C05477=1176.105,271.034,-67.370,-177.096,7.526,148.586
C05478=1176.109,270.786,-67.343,-177.099,7.524,148.586
C05479=1176.114,270.537,-67.314,-177.101,7.521,148.586
C05480=1176.118,270.290,-67.286,-177.104,7.518,148.586
C05481=1176.123,270.041,-67.257,-177.107,7.515,148.586
C05482=1176.127,269.793,-67.230,-177.109,7.513,148.586
C05483=1176.131,269.544,-67.202,-177.112,7.510,148.586
C05484=1176.135,269.295,-67.173,-177.114,7.507,148.586
C05485=1176.140,269.047,-67.145,-177.117,7.504,148.586
C05486=1176.144,268.799,-67.116,-177.119,7.502,148.586
C05487=1176.149,268.551,-67.088,-177.122,7.499,148.586
C05488=1176.153,268.302,-67.060,-177.125,7.496,148.586
C05489=1176.157,268.054,-67.032,-177.128,7.493,148.586
C05490=1176.162,267.806,-67.004,-177.130,7.491,148.586
C05491=1176.166,267.557,-66.975,-177.132,7.488,148.586
C05492=1176.171,267.309,-66.948,-177.136,7.485,148.587
C05493=1176.174,267.061,-66.920,-177.138,7.483,148.587
C05494=1176.180,266.812,-66.892,-177.141,7.480,148.587
C05495=1176.183,266.563,-66.864,-177.143,7.477,148.587
C05496=1176.188,266.315,-66.836,-177.146,7.474,148.587
C05497=1176.192,266.067,-66.807,-177.148,7.472,148.587
C05498=1176.197,265.819,-66.779,-177.151,7.469,148.587
C05499=1176.200,265.570,-66.751,-177.154,7.466,148.587
C05500=1176.206,265.321,-66.724,-177.156,7.463,148.587
C05501=1176.210,265.073,-66.696,-177.159,7.461,148.587
C05502=1176.214,264.825,-66.668,-177.161,7.458,148.587
C05503=1176.218,264.577,-66.640,-177.164,7.455,148.587
C05504=1176.223,264.327,-66.612,-177.167,7.453,148.588
C05505=1176.227,264.080,-66.584,-177.169,7.450,148.588
C05506=1176.232,263.832,-66.556,-177.172,7.447,148.588
C05507=1176.235,263.583,-66.528,-177.174,7.445,148.588
C05508=1176.241,263.334,-66.501,-177.177,7.442,148.588
C05509=1176.245,263.086,-66.472,-177.180,7.439,148.588
C05510=1176.249,262.838,-66.445,-177.183,7.436,148.588
C05511=1176.254,262.565,-66.414,-177.185,7.433,148.588
C05512=1176.259,262.292,-66.384,-177.189,7.430,148.588
C05513=1176.264,262.019,-66.353,-177.191,7.427,148.588
C05514=1176.268,261.745,-66.322,-177.194,7.424,148.588
C05515=1176.273,261.497,-66.295,-177.197,7.421,148.589
C05516=1176.277,261.249,-66.267,-177.199,7.419,148.589
C05517=1176.281,261.000,-66.239,-177.202,7.417,148.589
C05518=1176.286,260.752,-66.212,-177.205,7.414,148.589
C05519=1176.290,260.504,-66.184,-177.207,7.412,148.589
C05520=1176.295,260.254,-66.156,-177.210,7.409,148.589
C05521=1176.299,260.007,-66.129,-177.213,7.406,148.589
C05522=1176.304,259.758,-66.102,-177.215,7.403,148.589
C05523=1176.308,259.509,-66.073,-177.217,7.400,148.589
C05524=1176.312,259.261,-66.046,-177.221,7.398,148.590
C05525=1176.317,259.013,-66.019,-177.223,7.396,148.590
C05526=1176.321,258.765,-65.992,-177.226,7.393,148.590
C05527=1176.325,258.516,-65.963,-177.228,7.390,148.590
C05528=1176.330,258.268,-65.936,-177.231,7.388,148.590
C05529=1176.334,258.019,-65.909,-177.233,7.385,148.590
C05530=1176.338,257.770,-65.881,-177.236,7.382,148.590
C05531=1176.343,257.522,-65.854,-177.239,7.380,148.590
C05532=1176.347,257.274,-65.826,-177.241,7.377,148.590
C05533=1176.352,257.026,-65.799,-177.244,7.374,148.590
C05534=1176.356,256.776,-65.772,-177.246,7.372,148.590
C05535=1176.360,256.529,-65.744,-177.249,7.369,148.591
C05536=1176.365,256.280,-65.717,-177.252,7.366,148.591
C05537=1176.369,256.032,-65.690,-177.254,7.364,148.591
C05538=1176.373,255.783,-65.662,-177.257,7.361,148.591
C05539=1176.378,255.534,-65.635,-177.260,7.358,148.591
C05540=1176.382,255.286,-65.608,-177.262,7.356,148.591
C05541=1176.387,255.038,-65.580,-177.265,7.353,148.591
C05542=1176.391,254.789,-65.552,-177.268,7.350,148.591
C05543=1176.396,254.540,-65.525,-177.270,7.348,148.592
C05544=1176.400,254.292,-65.498,-177.273,7.345,148.592
C05545=1176.405,254.044,-65.471,-177.276,7.342,148.592
C05546=1176.409,253.796,-65.444,-177.278,7.340,148.592
C05547=1176.413,253.546,-65.416,-177.281,7.337,148.592
C05548=1176.418,253.298,-65.389,-177.283,7.335,148.592
C05549=1176.422,253.050,-65.363,-177.286,7.332,148.592
C05550=1176.426,252.801,-65.336,-177.289,7.330,148.592
C05551=1176.431,252.553,-65.308,-177.291,7.327,148.593
C05552=1176.436,252.305,-65.281,-177.294,7.325,148.593
C05553=1176.440,252.056,-65.253,-177.297,7.322,148.593
C05554=1176.444,251.807,-65.226,-177.299,7.319,148.593
C05555=1176.449,251.559,-65.199,-177.302,7.317,148.593
C05556=1176.453,251.310,-65.173,-177.304,7.315,148.593
C05557=1176.457,251.062,-65.146,-177.307,7.312,148.593
C05558=1176.462,250.813,-65.119,-177.310,7.309,148.593
C05559=1176.467,250.565,-65.091,-177.313,7.307,148.594
C05560=1176.471,250.316,-65.064,-177.315,7.304,148.594
C05561=1176.475,250.068,-65.038,-177.318,7.301,148.594
C05562=1176.479,249.819,-65.011,-177.320,7.299,148.594
C05563=1176.484,249.571,-64.983,-177.323,7.296,148.594
C05564=1176.489,249.322,-64.956,-177.326,7.294,148.594
C05565=1176.493,249.074,-64.930,-177.328,7.291,148.594
C05566=1176.497,248.825,-64.903,-177.331,7.288,148.594
C05567=1176.502,248.577,-64.876,-177.334,7.286,148.595
C05568=1176.507,248.328,-64.849,-177.337,7.283,148.595
C05569=1176.510,248.080,-64.822,-177.339,7.281,148.595
C05570=1176.515,247.831,-64.795,-177.342,7.278,148.595
C05571=1176.519,247.583,-64.768,-177.345,7.276,148.595
C05572=1176.523,247.334,-64.741,-177.347,7.273,148.595
C05573=1176.528,247.086,-64.714,-177.350,7.270,148.595
C05574=1176.533,246.837,-64.688,-177.352,7.269,148.596
C05575=1176.537,246.589,-64.661,-177.355,7.266,148.596
C05576=1176.541,246.340,-64.634,-177.358,7.263,148.596
C05577=1176.546,246.092,-64.607,-177.360,7.261,148.596
C05578=1176.550,245.843,-64.581,-177.363,7.258,148.596
C05579=1176.555,245.595,-64.554,-177.365,7.256,148.596
C05580=1176.560,245.346,-64.527,-177.368,7.253,148.596
C05581=1176.563,245.098,-64.501,-177.371,7.251,148.597
C05582=1176.568,244.849,-64.474,-177.373,7.248,148.597
C05583=1176.572,244.601,-64.447,-177.376,7.245,148.597
C05584=1176.577,244.352,-64.421,-177.379,7.243,148.597
C05585=1176.582,244.103,-64.394,-177.382,7.240,148.597
C05586=1176.586,243.855,-64.368,-177.384,7.238,148.597
C05587=1176.590,243.607,-64.341,-177.387,7.235,148.597
C05588=1176.594,243.358,-64.315,-177.389,7.233,148.598
C05589=1176.599,243.109,-64.288,-177.392,7.230,148.598
C05590=1176.603,242.861,-64.261,-177.395,7.228,148.598
C05591=1176.608,242.612,-64.235,-177.397,7.226,148.598
C05592=1176.612,242.364,-64.208,-177.400,7.223,148.598
C05593=1176.617,242.115,-64.182,-177.403,7.221,148.598
C05594=1176.622,241.866,-64.155,-177.405,7.218,148.598
C05595=1176.625,241.618,-64.129,-177.408,7.216,148.599
C05596=1176.630,241.369,-64.102,-177.411,7.213,148.599
C05597=1176.634,241.121,-64.076,-177.413,7.211,148.599
C05598=1176.639,240.872,-64.050,-177.416,7.208,148.599
C05599=1176.643,240.623,-64.023,-177.419,7.205,148.599
C05600=1176.647,240.375,-63.997,-177.421,7.203,148.599
C05601=1176.653,240.127,-63.970,-177.424,7.200,148.600
C05602=1176.657,239.878,-63.945,-177.427,7.198,148.600
C05603=1176.662,239.630,-63.918,-177.429,7.195,148.600
C05604=1176.666,239.381,-63.892,-177.432,7.194,148.600
C05605=1176.670,239.132,-63.865,-177.435,7.191,148.600
C05606=1176.675,238.883,-63.839,-177.437,7.189,148.600
C05607=1176.679,238.635,-63.813,-177.440,7.186,148.601
C05608=1176.684,238.386,-63.786,-177.442,7.184,148.601
C05609=1176.687,238.138,-63.760,-177.445,7.181,148.601
C05610=1176.692,237.889,-63.733,-177.448,7.179,148.601
C05611=1176.697,237.641,-63.708,-177.450,7.176,148.601
C05612=1176.701,237.393,-63.682,-177.453,7.174,148.602
C05613=1176.706,237.143,-63.655,-177.456,7.171,148.602
C05614=1176.710,236.895,-63.629,-177.459,7.168,148.602
C05615=1176.715,236.623,-63.601,-177.461,7.166,148.602
C05616=1176.720,236.352,-63.571,-177.464,7.164,148.602
C05617=1176.725,236.080,-63.543,-177.467,7.161,148.602
C05618=1176.730,235.809,-63.515,-177.470,7.158,148.603
C05619=1176.735,235.560,-63.489,-177.473,7.156,148.603
C05620=1176.739,235.311,-63.463,-177.475,7.153,148.603
C05621=1176.743,235.063,-63.437,-177.478,7.151,148.603
C05622=1176.748,234.814,-63.410,-177.481,7.148,148.603
C05623=1176.752,234.565,-63.384,-177.483,7.147,148.604
C05624=1176.757,234.317,-63.359,-177.486,7.144,148.604
C05625=1176.761,234.068,-63.333,-177.488,7.141,148.604
C05626=1176.766,233.820,-63.306,-177.492,7.139,148.604
C05627=1176.770,233.571,-63.280,-177.494,7.137,148.604
C05628=1176.775,233.323,-63.255,-177.497,7.134,148.604
C05629=1176.779,233.074,-63.229,-177.499,7.132,148.605
C05630=1176.784,232.825,-63.203,-177.502,7.129,148.605
C05631=1176.788,232.576,-63.177,-177.505,7.127,148.605
C05632=1176.792,232.328,-63.151,-177.508,7.125,148.605
C05633=1176.797,232.080,-63.125,-177.510,7.122,148.605
C05634=1176.801,231.831,-63.100,-177.513,7.119,148.605
C05635=1176.805,231.582,-63.074,-177.515,7.118,148.606
C05636=1176.810,231.333,-63.047,-177.518,7.115,148.606
C05637=1176.815,231.085,-63.022,-177.521,7.113,148.606
C05638=1176.819,230.836,-62.996,-177.523,7.110,148.606
C05639=1176.823,230.587,-62.971,-177.526,7.108,148.607
C05640=1176.828,230.339,-62.945,-177.529,7.105,148.607
C05641=1176.833,230.091,-62.919,-177.532,7.103,148.607
C05642=1176.837,229.841,-62.893,-177.534,7.100,148.607
C05643=1176.842,229.593,-62.867,-177.537,7.099,148.607
C05644=1176.847,229.345,-62.842,-177.540,7.096,148.607
C05645=1176.851,229.096,-62.816,-177.542,7.094,148.608
C05646=1176.855,228.847,-62.790,-177.545,7.092,148.608
C05647=1176.860,228.599,-62.765,-177.548,7.089,148.608
C05648=1176.864,228.350,-62.739,-177.550,7.087,148.608
C05649=1176.868,228.101,-62.714,-177.553,7.084,148.608
C05650=1176.873,227.853,-62.688,-177.555,7.082,148.609
C05651=1176.877,227.604,-62.662,-177.558,7.079,148.609
C05652=1176.882,227.355,-62.637,-177.561,7.077,148.609
C05653=1176.886,227.107,-62.611,-177.564,7.074,148.609
C05654=1176.891,226.858,-62.586,-177.566,7.073,148.610
C05655=1176.895,226.609,-62.561,-177.569,7.070,148.610
C05656=1176.900,226.361,-62.535,-177.572,7.068,148.610
C05657=1176.904,226.112,-62.509,-177.574,7.066,148.610
C05658=1176.908,225.863,-62.484,-177.577,7.063,148.610
C05659=1176.913,225.615,-62.458,-177.579,7.061,148.610
C05660=1176.918,225.366,-62.433,-177.582,7.058,148.611
C05661=1176.922,225.117,-62.407,-177.585,7.056,148.611
C05662=1176.927,224.869,-62.382,-177.588,7.054,148.611
C05663=1176.931,224.620,-62.356,-177.590,7.052,148.611
C05664=1176.936,224.371,-62.332,-177.593,7.050,148.612
C05665=1176.940,224.123,-62.306,-177.596,7.047,148.612
C05666=1176.945,223.874,-62.280,-177.598,7.045,148.612
C05667=1176.949,223.626,-62.255,-177.601,7.042,148.612
C05668=1176.954,223.376,-62.230,-177.603,7.040,148.612
C05669=1176.959,223.128,-62.204,-177.607,7.037,148.613
C05670=1176.963,222.879,-62.179,-177.609,7.035,148.613
C05671=1176.967,222.631,-62.155,-177.612,7.034,148.613
C05672=1176.972,222.382,-62.129,-177.614,7.031,148.613
C05673=1176.976,222.133,-62.103,-177.617,7.029,148.614
C05674=1176.981,221.885,-62.078,-177.620,7.026,148.614
C05675=1176.985,221.636,-62.053,-177.622,7.024,148.614
C05676=1176.990,221.387,-62.028,-177.625,7.022,148.614
C05677=1176.995,221.138,-62.002,-177.628,7.019,148.614
C05678=1176.999,220.891,-61.977,-177.630,7.017,148.615
C05679=1177.003,220.641,-61.952,-177.633,7.014,148.615
C05680=1177.008,220.393,-61.927,-177.636,7.013,148.615
C05681=1177.013,220.144,-61.902,-177.638,7.011,148.615
C05682=1177.017,219.896,-61.877,-177.641,7.008,148.616
C05683=1177.021,219.646,-61.852,-177.644,7.006,148.616
C05684=1177.026,219.398,-61.827,-177.647,7.003,148.616
C05685=1177.031,219.149,-61.802,-177.649,7.001,148.616
C05686=1177.035,218.901,-61.776,-177.652,6.999,148.616
C05687=1177.040,218.651,-61.751,-177.655,6.997,148.617
C05688=1177.044,218.404,-61.726,-177.657,6.994,148.617
C05689=1177.048,218.154,-61.701,-177.660,6.992,148.617
C05690=1177.053,217.906,-61.676,-177.663,6.990,148.618
C05691=1177.057,217.657,-61.652,-177.665,6.988,148.618
C05692=1177.062,217.408,-61.627,-177.668,6.985,148.618
C05693=1177.066,217.159,-61.601,-177.670,6.983,148.618
C05694=1177.072,216.911,-61.577,-177.674,6.981,148.618
C05695=1177.075,216.662,-61.551,-177.676,6.979,148.619
C05696=1177.080,216.413,-61.527,-177.678,6.977,148.619
C05697=1177.085,216.164,-61.502,-177.682,6.974,148.619
C05698=1177.089,215.916,-61.477,-177.684,6.972,148.619
C05699=1177.093,215.667,-61.452,-177.687,6.970,148.620
C05700=1177.098,215.418,-61.427,-177.690,6.967,148.620
C05701=1177.103,215.170,-61.402,-177.692,6.965,148.620
C05702=1177.107,214.921,-61.377,-177.695,6.964,148.620
C05703=1177.112,214.672,-61.353,-177.697,6.961,148.620
C05704=1177.116,214.423,-61.328,-177.700,6.959,148.621
C05705=1177.121,214.175,-61.303,-177.703,6.956,148.621
C05706=1177.125,213.927,-61.279,-177.705,6.954,148.621
C05707=1177.130,213.677,-61.254,-177.708,6.952,148.622
C05708=1177.135,213.428,-61.229,-177.711,6.949,148.622
C05709=1177.138,213.180,-61.204,-177.714,6.947,148.622
C05710=1177.144,212.931,-61.179,-177.716,6.946,148.622
C05711=1177.148,212.683,-61.155,-177.719,6.943,148.622
C05712=1177.152,212.433,-61.130,-177.722,6.941,148.623
C05713=1177.157,212.185,-61.106,-177.724,6.939,148.623
C05714=1177.162,211.936,-61.081,-177.727,6.936,148.623
C05715=1177.165,211.688,-61.056,-177.730,6.934,148.623
C05716=1177.171,211.439,-61.032,-177.732,6.932,148.624
C05717=1177.176,211.190,-61.007,-177.735,6.930,148.624
C05718=1177.180,210.941,-60.982,-177.738,6.928,148.624
C05719=1177.185,210.671,-60.956,-177.741,6.925,148.625
C05720=1177.190,210.401,-60.929,-177.743,6.923,148.625
C05721=1177.195,210.129,-60.903,-177.746,6.920,148.625
C05722=1177.200,209.859,-60.876,-177.750,6.918,148.625
C05723=1177.204,209.611,-60.852,-177.752,6.916,148.626
C05724=1177.209,209.361,-60.827,-177.755,6.914,148.626
C05725=1177.213,209.113,-60.803,-177.758,6.911,148.626
C05726=1177.218,208.864,-60.778,-177.760,6.910,148.626
C05727=1177.222,208.615,-60.754,-177.763,6.907,148.627
C05728=1177.226,208.367,-60.730,-177.765,6.906,148.627
C05729=1177.232,208.118,-60.705,-177.768,6.903,148.627
C05730=1177.236,207.869,-60.681,-177.771,6.901,148.627
C05731=1177.241,207.620,-60.656,-177.773,6.899,148.628
C05732=1177.245,207.372,-60.632,-177.776,6.896,148.628
C05733=1177.250,207.123,-60.607,-177.779,6.894,148.628
C05734=1177.254,206.874,-60.583,-177.781,6.893,148.628
C05735=1177.258,206.625,-60.559,-177.785,6.890,148.629
C05736=1177.263,206.377,-60.534,-177.787,6.888,148.629
C05737=1177.268,206.128,-60.510,-177.790,6.886,148.629
C05738=1177.272,205.879,-60.486,-177.793,6.883,148.630
C05739=1177.277,205.630,-60.461,-177.795,6.881,148.630
C05740=1177.281,205.381,-60.437,-177.798,6.879,148.630
C05741=1177.286,205.133,-60.413,-177.800,6.878,148.630
C05742=1177.291,204.884,-60.389,-177.803,6.875,148.630
C05743=1177.296,204.635,-60.365,-177.806,6.873,148.631
C05744=1177.299,204.386,-60.341,-177.808,6.871,148.631
C05745=1177.305,204.137,-60.316,-177.811,6.868,148.631
C05746=1177.309,203.889,-60.292,-177.814,6.866,148.632
C05747=1177.313,203.641,-60.268,-177.816,6.865,148.632
C05748=1177.318,203.392,-60.245,-177.819,6.862,148.632
C05749=1177.323,203.142,-60.220,-177.822,6.860,148.632
C05750=1177.327,202.894,-60.196,-177.825,6.858,148.633
C05751=1177.332,202.645,-60.172,-177.827,6.856,148.633
C05752=1177.336,202.396,-60.148,-177.830,6.853,148.633
C05753=1177.341,202.148,-60.123,-177.833,6.852,148.633
C05754=1177.345,201.898,-60.100,-177.835,6.850,148.634
C05755=1177.350,201.649,-60.076,-177.838,6.848,148.634
C05756=1177.354,201.401,-60.052,-177.841,6.845,148.634
C05757=1177.360,201.152,-60.028,-177.843,6.843,148.635
C05758=1177.364,200.903,-60.004,-177.846,6.841,148.635
C05759=1177.368,200.655,-59.979,-177.848,6.839,148.635
C05760=1177.373,200.406,-59.956,-177.852,6.837,148.635
C05761=1177.377,200.157,-59.932,-177.854,6.835,148.636
C05762=1177.381,199.908,-59.908,-177.856,6.833,148.636
C05763=1177.387,199.659,-59.884,-177.859,6.831,148.636
C05764=1177.391,199.410,-59.860,-177.862,6.828,148.637
C05765=1177.396,199.161,-59.836,-177.865,6.827,148.637
C05766=1177.400,198.913,-59.812,-177.867,6.824,148.637
C05767=1177.405,198.664,-59.789,-177.870,6.823,148.637
C05768=1177.409,198.416,-59.765,-177.873,6.820,148.638
C05769=1177.414,198.167,-59.741,-177.876,6.818,148.638
C05770=1177.418,197.918,-59.717,-177.878,6.816,148.638
C05771=1177.423,197.668,-59.693,-177.881,6.814,148.639
C05772=1177.428,197.419,-59.670,-177.884,6.812,148.639
C05773=1177.432,197.171,-59.645,-177.887,6.810,148.639
C05774=1177.437,196.922,-59.622,-177.889,6.808,148.639
C05775=1177.441,196.673,-59.598,-177.891,6.806,148.640
C05776=1177.446,196.424,-59.575,-177.895,6.803,148.640
C05777=1177.450,196.176,-59.551,-177.897,6.802,148.640
C05778=1177.455,195.927,-59.527,-177.899,6.800,148.640
C05779=1177.460,195.678,-59.504,-177.902,6.798,148.641
C05780=1177.464,195.429,-59.480,-177.905,6.795,148.641
C05781=1177.469,195.180,-59.456,-177.908,6.793,148.642
C05782=1177.474,194.931,-59.433,-177.910,6.791,148.642
C05783=1177.478,194.683,-59.409,-177.913,6.789,148.642
C05784=1177.483,194.434,-59.386,-177.916,6.788,148.642
C05785=1177.487,194.185,-59.362,-177.919,6.785,148.643
C05786=1177.492,193.936,-59.338,-177.921,6.783,148.643
C05787=1177.497,193.687,-59.315,-177.924,6.781,148.643
C05788=1177.501,193.438,-59.292,-177.926,6.779,148.643
C05789=1177.506,193.189,-59.268,-177.929,6.778,148.644
C05790=1177.510,192.941,-59.244,-177.932,6.775,148.644
C05791=1177.515,192.692,-59.221,-177.934,6.773,148.644
C05792=1177.520,192.443,-59.197,-177.937,6.771,148.645
C05793=1177.524,192.194,-59.174,-177.940,6.769,148.645
C05794=1177.529,191.945,-59.150,-177.943,6.767,148.645
C05795=1177.533,191.697,-59.127,-177.946,6.765,148.646
C05796=1177.537,191.448,-59.104,-177.948,6.763,148.646
C05797=1177.542,191.199,-59.080,-177.951,6.761,148.646
C05798=1177.547,190.949,-59.057,-177.953,6.759,148.647
C05799=1177.552,190.700,-59.034,-177.957,6.757,148.647
C05800=1177.556,190.452,-59.010,-177.959,6.755,148.647
C05801=1177.561,190.203,-58.986,-177.961,6.753,148.647
C05802=1177.566,189.955,-58.963,-177.964,6.751,148.648
C05803=1177.571,189.706,-58.940,-177.967,6.749,148.648
C05804=1177.575,189.457,-58.917,-177.969,6.747,148.648
C05805=1177.579,189.208,-58.894,-177.973,6.745,148.649
C05806=1177.584,188.959,-58.870,-177.975,6.743,148.649
C05807=1177.589,188.710,-58.847,-177.978,6.741,148.649
C05808=1177.593,188.461,-58.824,-177.980,6.739,148.650
C05809=1177.597,188.212,-58.801,-177.983,6.737,148.650
C05810=1177.602,187.963,-58.778,-177.986,6.735,148.650
C05811=1177.607,187.714,-58.754,-177.988,6.733,148.650
C05812=1177.612,187.466,-58.731,-177.991,6.731,148.651
C05813=1177.617,187.217,-58.708,-177.994,6.729,148.651
C05814=1177.621,186.968,-58.685,-177.996,6.727,148.651
C05815=1177.625,186.719,-58.662,-177.999,6.725,148.652
C05816=1177.630,186.470,-58.638,-178.002,6.723,148.652
C05817=1177.635,186.221,-58.615,-178.004,6.721,148.652
C05818=1177.639,185.972,-58.592,-178.007,6.719,148.653
C05819=1177.644,185.724,-58.569,-178.010,6.717,148.653
C05820=1177.649,185.475,-58.546,-178.012,6.715,148.653
C05821=1177.653,185.226,-58.523,-178.015,6.714,148.654
C05822=1177.658,184.976,-58.501,-178.018,6.712,148.654
C05823=1177.663,184.707,-58.475,-178.021,6.709,148.654
C05824=1177.667,184.438,-58.450,-178.024,6.707,148.655
C05825=1177.673,184.168,-58.425,-178.027,6.705,148.655
C05826=1177.678,183.898,-58.400,-178.030,6.703,148.655
C05827=1177.682,183.650,-58.378,-178.032,6.701,148.656
C05828=1177.687,183.400,-58.354,-178.035,6.699,148.656
C05829=1177.692,183.152,-58.332,-178.038,6.697,148.656
C05830=1177.696,182.903,-58.309,-178.040,6.695,148.657
C05831=1177.701,182.654,-58.286,-178.043,6.693,148.657
C05832=1177.706,182.405,-58.262,-178.046,6.691,148.657
C05833=1177.710,182.155,-58.240,-178.048,6.689,148.658
C05834=1177.715,181.907,-58.217,-178.051,6.687,148.658
C05835=1177.719,181.658,-58.195,-178.053,6.686,148.658
C05836=1177.724,181.409,-58.171,-178.056,6.684,148.659
C05837=1177.728,181.160,-58.149,-178.059,6.681,148.659
C05838=1177.733,180.912,-58.126,-178.062,6.679,148.659
C05839=1177.738,180.663,-58.103,-178.065,6.678,148.660
C05840=1177.742,180.413,-58.081,-178.067,6.676,148.660
C05841=1177.747,180.164,-58.057,-178.070,6.674,148.660
C05842=1177.752,179.916,-58.035,-178.072,6.672,148.660
C05843=1177.757,179.667,-58.012,-178.075,6.670,148.661
C05844=1177.761,179.418,-57.990,-178.078,6.668,148.661
C05845=1177.765,179.169,-57.966,-178.081,6.666,148.662
C05846=1177.770,178.920,-57.945,-178.083,6.664,148.662
C05847=1177.775,178.671,-57.921,-178.086,6.662,148.662
C05848=1177.779,178.422,-57.899,-178.089,6.661,148.663
C05849=1177.784,178.173,-57.876,-178.091,6.659,148.663
C05850=1177.789,177.924,-57.854,-178.094,6.657,148.663
C05851=1177.793,177.675,-57.831,-178.096,6.655,148.663
C05852=1177.798,177.427,-57.808,-178.099,6.653,148.664
C05853=1177.803,177.177,-57.786,-178.102,6.651,148.664
C05854=1177.807,176.929,-57.763,-178.104,6.650,148.665
C05855=1177.813,176.680,-57.741,-178.108,6.647,148.665
C05856=1177.817,176.431,-57.718,-178.110,6.645,148.665
C05857=1177.821,176.182,-57.696,-178.113,6.643,148.666
C05858=1177.826,175.933,-57.674,-178.116,6.642,148.666
C05859=1177.830,175.684,-57.651,-178.118,6.640,148.666
C05860=1177.835,175.434,-57.628,-178.121,6.638,148.666
C05861=1177.840,175.186,-57.606,-178.123,6.636,148.667
C05862=1177.845,174.937,-57.583,-178.126,6.634,148.667
C05863=1177.849,174.688,-57.560,-178.129,6.632,148.668
C05864=1177.854,174.439,-57.539,-178.131,6.631,148.668
C05865=1177.859,174.190,-57.516,-178.134,6.629,148.668
C05866=1177.863,173.941,-57.493,-178.137,6.627,148.669
C05867=1177.868,173.692,-57.472,-178.140,6.624,148.669
C05868=1177.872,173.443,-57.448,-178.143,6.623,148.669
C05869=1177.877,173.195,-57.427,-178.145,6.621,148.670
C05870=1177.881,172.945,-57.405,-178.148,6.619,148.670
C05871=1177.886,172.696,-57.381,-178.151,6.617,148.670
C05872=1177.891,172.448,-57.359,-178.153,6.616,148.671
C05873=1177.895,172.198,-57.337,-178.156,6.614,148.671
C05874=1177.901,171.949,-57.315,-178.158,6.612,148.671
C05875=1177.905,171.701,-57.292,-178.161,6.610,148.672
C05876=1177.910,171.452,-57.271,-178.164,6.608,148.672
C05877=1177.915,171.202,-57.248,-178.166,6.606,148.672
C05878=1177.919,170.953,-57.226,-178.169,6.605,148.673
C05879=1177.924,170.705,-57.204,-178.172,6.603,148.673
C05880=1177.928,170.456,-57.182,-178.174,6.601,148.674
C05881=1177.933,170.207,-57.159,-178.177,6.599,148.674
C05882=1177.938,169.957,-57.137,-178.180,6.598,148.674
C05883=1177.943,169.709,-57.116,-178.182,6.596,148.675
C05884=1177.947,169.460,-57.093,-178.186,6.593,148.675
C05885=1177.952,169.211,-57.071,-178.188,6.591,148.675
C05886=1177.956,168.962,-57.048,-178.191,6.590,148.676
C05887=1177.961,168.713,-57.027,-178.194,6.588,148.676
C05888=1177.966,168.464,-57.005,-178.196,6.586,148.676
C05889=1177.970,168.215,-56.983,-178.199,6.584,148.677
C05890=1177.975,167.965,-56.960,-178.202,6.583,148.677
C05891=1177.980,167.717,-56.938,-178.204,6.581,148.678
C05892=1177.984,167.468,-56.916,-178.207,6.579,148.678
C05893=1177.989,167.219,-56.894,-178.210,6.577,148.678
C05894=1177.993,166.970,-56.872,-178.212,6.576,148.679
C05895=1177.998,166.721,-56.851,-178.215,6.574,148.679
C05896=1178.003,166.472,-56.829,-178.217,6.572,148.679
C05897=1178.008,166.223,-56.806,-178.220,6.570,148.680
C05898=1178.012,165.974,-56.784,-178.223,6.568,148.680
C05899=1178.017,165.725,-56.763,-178.225,6.566,148.680
C05900=1178.022,165.476,-56.740,-178.228,6.565,148.681
C05901=1178.026,165.227,-56.719,-178.231,6.563,148.681
C05902=1178.031,164.979,-56.697,-178.233,6.561,148.681
C05903=1178.036,164.729,-56.675,-178.236,6.559,148.682
C05904=1178.040,164.481,-56.653,-178.239,6.558,148.682
C05905=1178.045,164.231,-56.631,-178.241,6.556,148.682
C05906=1178.050,163.983,-56.610,-178.244,6.554,148.683
C05907=1178.054,163.733,-56.588,-178.247,6.552,148.683
C05908=1178.059,163.484,-56.567,-178.249,6.550,148.684
C05909=1178.064,163.234,-56.544,-178.252,6.549,148.684
C05910=1178.069,162.986,-56.522,-178.255,6.547,148.684
C05911=1178.074,162.737,-56.501,-178.258,6.545,148.685
C05912=1178.078,162.488,-56.479,-178.260,6.543,148.685
C05913=1178.083,162.239,-56.457,-178.263,6.542,148.685
C05914=1178.087,161.990,-56.435,-178.266,6.540,148.686
C05915=1178.092,161.741,-56.413,-178.268,6.538,148.686
C05916=1178.097,161.492,-56.392,-178.271,6.536,148.687
C05917=1178.101,161.242,-56.370,-178.274,6.535,148.687
C05918=1178.106,160.994,-56.349,-178.276,6.533,148.687
C05919=1178.110,160.746,-56.327,-178.279,6.531,148.688
C05920=1178.115,160.496,-56.305,-178.282,6.529,148.688
C05921=1178.120,160.247,-56.284,-178.284,6.528,148.688
C05922=1178.125,159.998,-56.263,-178.287,6.526,148.689
C05923=1178.129,159.749,-56.241,-178.290,6.524,148.689
C05924=1178.134,159.500,-56.220,-178.292,6.522,148.690
C05925=1178.139,159.251,-56.198,-178.296,6.521,148.690
C05926=1178.143,159.002,-56.176,-178.298,6.519,148.691
C05927=1178.148,158.733,-56.153,-178.301,6.517,148.691
C05928=1178.153,158.464,-56.129,-178.304,6.516,148.691
C05929=1178.158,158.195,-56.106,-178.306,6.514,148.692
C05930=1178.164,157.925,-56.083,-178.310,6.511,148.692
C05931=1178.168,157.677,-56.061,-178.312,6.509,148.692
C05932=1178.174,157.428,-56.040,-178.314,6.508,148.693
C05933=1178.178,157.179,-56.019,-178.317,6.507,148.693
C05934=1178.182,156.930,-55.997,-178.320,6.505,148.694
C05935=1178.187,156.681,-55.976,-178.323,6.504,148.694
C05936=1178.192,156.432,-55.955,-178.326,6.502,148.694
C05937=1178.197,156.182,-55.933,-178.328,6.500,148.695
C05938=1178.201,155.933,-55.912,-178.331,6.498,148.695
C05939=1178.207,155.684,-55.891,-178.334,6.496,148.696
C05940=1178.211,155.436,-55.869,-178.336,6.495,148.696
C05941=1178.215,155.186,-55.847,-178.339,6.493,148.696
C05942=1178.220,154.937,-55.826,-178.342,6.491,148.697
C05943=1178.225,154.689,-55.805,-178.344,6.489,148.697
C05944=1178.230,154.439,-55.784,-178.347,6.488,148.698
C05945=1178.234,154.190,-55.762,-178.350,6.486,148.698
C05946=1178.239,153.941,-55.741,-178.353,6.484,148.698
C05947=1178.244,153.692,-55.720,-178.355,6.482,148.699
C05948=1178.249,153.443,-55.699,-178.358,6.481,148.699
C05949=1178.253,153.194,-55.677,-178.361,6.479,148.699
C05950=1178.258,152.945,-55.656,-178.363,6.478,148.700
C05951=1178.263,152.696,-55.635,-178.365,6.476,148.700
C05952=1178.268,152.447,-55.614,-178.369,6.475,148.701
C05953=1178.272,152.198,-55.593,-178.371,6.473,148.701
C05954=1178.276,151.949,-55.571,-178.374,6.471,148.702
C05955=1178.282,151.699,-55.550,-178.377,6.469,148.702
C05956=1178.286,151.450,-55.530,-178.379,6.468,148.702
C05957=1178.291,151.202,-55.508,-178.382,6.466,148.703
C05958=1178.296,150.953,-55.487,-178.385,6.464,148.703
C05959=1178.301,150.704,-55.467,-178.387,6.462,148.703
C05960=1178.305,150.454,-55.445,-178.390,6.461,148.704
C05961=1178.310,150.205,-55.424,-178.393,6.459,148.704
C05962=1178.314,149.956,-55.403,-178.395,6.458,148.705
C05963=1178.319,149.707,-55.382,-178.398,6.456,148.705
C05964=1178.324,149.458,-55.361,-178.401,6.455,148.706
C05965=1178.329,149.209,-55.340,-178.403,6.453,148.706
C05966=1178.333,148.960,-55.318,-178.406,6.451,148.706
C05967=1178.338,148.711,-55.298,-178.409,6.450,148.707
C05968=1178.343,148.462,-55.277,-178.412,6.448,148.707
C05969=1178.348,148.212,-55.256,-178.414,6.446,148.707
C05970=1178.352,147.964,-55.235,-178.417,6.444,148.708
C05971=1178.357,147.715,-55.214,-178.420,6.443,148.708
C05972=1178.362,147.466,-55.194,-178.422,6.442,148.709
C05973=1178.367,147.217,-55.173,-178.424,6.440,148.709
C05974=1178.371,146.967,-55.151,-178.428,6.438,148.710
C05975=1178.376,146.718,-55.131,-178.430,6.437,148.710
C05976=1178.381,146.469,-55.109,-178.433,6.435,148.710
C05977=1178.385,146.220,-55.089,-178.436,6.433,148.711
C05978=1178.390,145.971,-55.068,-178.438,6.431,148.711
C05979=1178.395,145.722,-55.048,-178.441,6.430,148.712
C05980=1178.400,145.473,-55.027,-178.444,6.428,148.712
C05981=1178.404,145.224,-55.006,-178.446,6.427,148.712
C05982=1178.410,144.974,-54.985,-178.449,6.425,148.713
C05983=1178.414,144.725,-54.965,-178.452,6.424,148.713
C05984=1178.419,144.477,-54.943,-178.454,6.422,148.714
C05985=1178.423,144.228,-54.923,-178.457,6.420,148.714
C05986=1178.428,143.979,-54.902,-178.460,6.419,148.714
C05987=1178.432,143.729,-54.881,-178.462,6.417,148.715
C05988=1178.437,143.480,-54.860,-178.465,6.416,148.715
C05989=1178.442,143.231,-54.840,-178.467,6.414,148.716
C05990=1178.446,142.982,-54.819,-178.470,6.412,148.716
C05991=1178.452,142.733,-54.799,-178.473,6.411,148.717
C05992=1178.456,142.484,-54.778,-178.476,6.409,148.717
C05993=1178.461,142.234,-54.757,-178.479,6.407,148.717
C05994=1178.466,141.985,-54.737,-178.481,6.406,148.718
C05995=1178.470,141.736,-54.716,-178.483,6.405,148.718
C05996=1178.475,141.487,-54.695,-178.486,6.403,148.719
C05997=1178.480,141.238,-54.675,-178.489,6.401,148.719
C05998=1178.485,140.989,-54.654,-178.492,6.400,148.720
C05999=1178.490,140.739,-54.634,-178.495,6.398,148.720
C06000=1178.494,140.490,-54.614,-178.497,6.396,148.720
C06001=1178.499,140.241,-54.593,-178.500,6.395,148.721
C06002=1178.504,139.992,-54.573,-178.502,6.394,148.721
C06003=1178.508,139.743,-54.552,-178.505,6.392,148.721
C06004=1178.513,139.494,-54.531,-178.508,6.391,148.722
C06005=1178.518,139.245,-54.511,-178.511,6.389,148.722
C06006=1178.522,138.996,-54.491,-178.513,6.387,148.723
C06007=1178.528,138.746,-54.470,-178.516,6.385,148.723
C06008=1178.533,138.498,-54.450,-178.518,6.384,148.724
C06009=1178.537,138.249,-54.430,-178.521,6.383,148.724
C06010=1178.542,138.000,-54.409,-178.524,6.381,148.724
C06011=1178.547,137.751,-54.389,-178.527,6.379,148.725
C06012=1178.551,137.501,-54.369,-178.529,6.378,148.725
C06013=1178.556,137.252,-54.349,-178.532,6.377,148.726
C06014=1178.561,137.003,-54.328,-178.534,6.375,148.726
C06015=1178.565,136.754,-54.307,-178.537,6.373,148.727
C06016=1178.570,136.505,-54.288,-178.540,6.372,148.727
C06017=1178.575,136.256,-54.267,-178.543,6.370,148.728
C06018=1178.580,136.006,-54.246,-178.546,6.368,148.728
C06019=1178.584,135.757,-54.226,-178.548,6.367,148.728
C06020=1178.589,135.508,-54.206,-178.550,6.366,148.729
C06021=1178.594,135.260,-54.186,-178.553,6.364,148.729
C06022=1178.599,135.010,-54.165,-178.556,6.363,148.730
C06023=1178.604,134.761,-54.146,-178.559,6.361,148.730
C06024=1178.608,134.512,-54.125,-178.561,6.360,148.731
C06025=1178.613,134.263,-54.105,-178.564,6.358,148.731
C06026=1178.618,134.013,-54.085,-178.566,6.356,148.731
C06027=1178.623,133.764,-54.064,-178.570,6.355,148.732
C06028=1178.628,133.515,-54.045,-178.572,6.353,148.732
C06029=1178.633,133.266,-54.025,-178.574,6.352,148.733
C06030=1178.637,133.017,-54.004,-178.577,6.351,148.733
C06031=1178.643,132.748,-53.983,-178.580,6.349,148.734
C06032=1178.648,132.480,-53.962,-178.583,6.347,148.734
C06033=1178.653,132.211,-53.939,-178.586,6.346,148.735
C06034=1178.658,131.943,-53.918,-178.589,6.344,148.735
C06035=1178.662,131.694,-53.898,-178.592,6.343,148.736
C06036=1178.667,131.444,-53.878,-178.594,6.341,148.736
C06037=1178.671,131.195,-53.858,-178.597,6.339,148.736
C06038=1178.676,130.946,-53.838,-178.599,6.338,148.737
C06039=1178.682,130.697,-53.817,-178.602,6.337,148.737
C06040=1178.687,130.448,-53.798,-178.605,6.335,148.738
C06041=1178.691,130.199,-53.777,-178.608,6.333,148.738
C06042=1178.696,129.949,-53.758,-178.610,6.332,148.739
C06043=1178.701,129.700,-53.738,-178.613,6.331,148.739
C06044=1178.706,129.451,-53.718,-178.616,6.329,148.740
C06045=1178.710,129.202,-53.698,-178.618,6.327,148.740
C06046=1178.715,128.953,-53.678,-178.621,6.327,148.740
C06047=1178.720,128.703,-53.658,-178.623,6.325,148.741
C06048=1178.725,128.455,-53.638,-178.626,6.323,148.741
C06049=1178.729,128.205,-53.619,-178.629,6.322,148.742
C06050=1178.734,127.956,-53.599,-178.631,6.321,148.742
C06051=1178.739,127.707,-53.579,-178.634,6.319,148.743
C06052=1178.744,127.458,-53.559,-178.637,6.318,148.743
C06053=1178.749,127.208,-53.540,-178.640,6.316,148.744
C06054=1178.753,126.959,-53.519,-178.642,6.315,148.744
C06055=1178.758,126.710,-53.500,-178.645,6.313,148.744
C06056=1178.763,126.461,-53.480,-178.647,6.311,148.745
C06057=1178.768,126.212,-53.460,-178.651,6.310,148.745
C06058=1178.772,125.962,-53.440,-178.653,6.309,148.746
C06059=1178.778,125.714,-53.421,-178.655,6.307,148.746
C06060=1178.782,125.464,-53.401,-178.658,6.306,148.747
C06061=1178.787,125.215,-53.381,-178.661,6.304,148.747
C06062=1178.791,124.966,-53.362,-178.663,6.303,148.748
C06063=1178.796,124.717,-53.343,-178.666,6.302,148.748
C06064=1178.801,124.467,-53.323,-178.669,6.300,148.748
C06065=1178.805,124.218,-53.303,-178.672,6.298,148.749
C06066=1178.811,123.970,-53.283,-178.674,6.298,148.749
C06067=1178.815,123.720,-53.264,-178.677,6.296,148.750
C06068=1178.820,123.470,-53.244,-178.680,6.294,148.750
C06069=1178.826,123.222,-53.225,-178.683,6.293,148.751
C06070=1178.830,122.973,-53.204,-178.685,6.292,148.751
C06071=1178.834,122.723,-53.185,-178.688,6.290,148.752
C06072=1178.839,122.474,-53.166,-178.690,6.288,148.752
C06073=1178.844,122.225,-53.146,-178.693,6.288,148.753
C06074=1178.849,121.975,-53.127,-178.696,6.286,148.753
C06075=1178.854,121.726,-53.107,-178.698,6.284,148.753
C06076=1178.859,121.477,-53.088,-178.701,6.283,148.754
C06077=1178.863,121.228,-53.068,-178.704,6.282,148.754
C06078=1178.868,120.979,-53.049,-178.706,6.280,148.755
C06079=1178.873,120.730,-53.029,-178.709,6.278,148.755
C06080=1178.878,120.481,-53.010,-178.712,6.278,148.756
C06081=1178.883,120.231,-52.990,-178.714,6.276,148.756
C06082=1178.887,119.982,-52.971,-178.717,6.274,148.757
C06083=1178.892,119.733,-52.952,-178.720,6.273,148.757
C06084=1178.897,119.484,-52.932,-178.722,6.272,148.758
C06085=1178.902,119.235,-52.913,-178.725,6.270,148.758
C06086=1178.906,118.986,-52.894,-178.728,6.269,148.759
C06087=1178.911,118.736,-52.874,-178.730,6.268,148.759
C06088=1178.916,118.487,-52.855,-178.733,6.266,148.760
C06089=1178.921,118.238,-52.835,-178.736,6.265,148.760
C06090=1178.926,117.989,-52.816,-178.738,6.264,148.760
C06091=1178.930,117.739,-52.797,-178.741,6.262,148.761
C06092=1178.935,117.490,-52.777,-178.744,6.261,148.761
C06093=1178.940,117.241,-52.758,-178.746,6.260,148.762
C06094=1178.944,116.992,-52.739,-178.749,6.258,148.762
C06095=1178.950,116.742,-52.720,-178.752,6.256,148.763
C06096=1178.955,116.493,-52.701,-178.754,6.256,148.763
C06097=1178.959,116.244,-52.682,-178.757,6.254,148.764
C06098=1178.964,115.995,-52.662,-178.760,6.252,148.764
C06099=1178.970,115.746,-52.643,-178.762,6.252,148.765
C06100=1178.974,115.496,-52.624,-178.765,6.250,148.765
C06101=1178.979,115.248,-52.605,-178.768,6.248,148.766
C06102=1178.984,114.998,-52.585,-178.771,6.247,148.766
C06103=1178.989,114.749,-52.567,-178.773,6.246,148.767
C06104=1178.993,114.499,-52.547,-178.776,6.244,148.767
C06105=1178.998,114.251,-52.529,-178.779,6.243,148.768
C06106=1179.003,114.001,-52.509,-178.781,6.242,148.768
C06107=1179.008,113.752,-52.490,-178.783,6.240,148.768
C06108=1179.012,113.502,-52.471,-178.786,6.239,148.769
C06109=1179.018,113.254,-52.452,-178.789,6.238,148.769
C06110=1179.022,113.004,-52.433,-178.791,6.236,148.770
C06111=1179.027,112.755,-52.414,-178.794,6.235,148.770
C06112=1179.032,112.505,-52.395,-178.797,6.234,148.771
C06113=1179.037,112.257,-52.376,-178.799,6.232,148.771
C06114=1179.041,112.007,-52.356,-178.802,6.231,148.772
C06115=1179.046,111.759,-52.338,-178.805,6.230,148.772
C06116=1179.051,111.508,-52.319,-178.808,6.228,148.773
C06117=1179.056,111.260,-52.300,-178.810,6.227,148.773
C06118=1179.060,111.010,-52.280,-178.813,6.226,148.774
C06119=1179.065,110.761,-52.262,-178.816,6.224,148.774
C06120=1179.071,110.512,-52.243,-178.818,6.223,148.775
C06121=1179.075,110.263,-52.224,-178.821,6.222,148.775
C06122=1179.080,110.013,-52.205,-178.824,6.220,148.776
C06123=1179.084,109.764,-52.186,-178.826,6.219,148.776
C06124=1179.090,109.515,-52.168,-178.829,6.218,148.777
C06125=1179.094,109.265,-52.149,-178.831,6.217,148.777
C06126=1179.099,109.017,-52.129,-178.834,6.215,148.778
C06127=1179.104,108.767,-52.111,-178.837,6.214,148.778
C06128=1179.109,108.518,-52.092,-178.839,6.213,148.779
C06129=1179.114,108.269,-52.074,-178.842,6.211,148.779
C06130=1179.119,108.019,-52.054,-178.845,6.210,148.780
C06131=1179.124,107.770,-52.036,-178.847,6.209,148.780
C06132=1179.129,107.521,-52.017,-178.850,6.207,148.781
C06133=1179.133,107.272,-51.998,-178.852,6.206,148.781
C06134=1179.138,107.023,-51.980,-178.855,6.205,148.781
C06135=1179.144,106.754,-51.960,-178.858,6.203,148.782
C06136=1179.149,106.485,-51.939,-178.861,6.202,148.782
C06137=1179.154,106.217,-51.919,-178.864,6.201,148.783
C06138=1179.159,105.949,-51.899,-178.867,6.200,148.784
C06139=1179.163,105.699,-51.880,-178.870,6.198,148.784
C06140=1179.168,105.451,-51.862,-178.872,6.196,148.785
C06141=1179.174,105.201,-51.843,-178.875,6.196,148.785
C06142=1179.178,104.951,-51.825,-178.878,6.194,148.786
C06143=1179.183,104.703,-51.805,-178.880,6.193,148.786
C06144=1179.188,104.453,-51.787,-178.883,6.192,148.787
C06145=1179.192,104.204,-51.768,-178.886,6.190,148.787
C06146=1179.198,103.955,-51.750,-178.888,6.189,148.788
C06147=1179.203,103.705,-51.732,-178.891,6.188,148.788
C06148=1179.207,103.456,-51.713,-178.893,6.187,148.789
C06149=1179.212,103.207,-51.694,-178.896,6.185,148.789
C06150=1179.217,102.957,-51.676,-178.898,6.184,148.790
C06151=1179.221,102.708,-51.657,-178.901,6.183,148.790
C06152=1179.226,102.459,-51.639,-178.904,6.181,148.791
C06153=1179.232,102.210,-51.621,-178.906,6.180,148.791
C06154=1179.237,101.961,-51.602,-178.909,6.179,148.791
C06155=1179.241,101.711,-51.584,-178.912,6.178,148.792
C06156=1179.247,101.462,-51.565,-178.915,6.176,148.793
C06157=1179.251,101.213,-51.546,-178.917,6.175,148.793
C06158=1179.255,100.963,-51.528,-178.920,6.174,148.794
C06159=1179.260,100.714,-51.510,-178.923,6.172,148.794
C06160=1179.266,100.465,-51.491,-178.925,6.172,148.795
C06161=1179.271,100.216,-51.473,-178.928,6.170,148.795
C06162=1179.275,99.966,-51.454,-178.930,6.169,148.795
C06163=1179.280,99.717,-51.436,-178.933,6.168,148.796
C06164=1179.285,99.468,-51.418,-178.936,6.166,148.797
C06165=1179.290,99.219,-51.399,-178.939,6.166,148.797
C06166=1179.294,98.969,-51.381,-178.941,6.164,148.798
C06167=1179.299,98.720,-51.363,-178.943,6.163,148.798
C06168=1179.304,98.471,-51.345,-178.947,6.162,148.799
C06169=1179.309,98.222,-51.327,-178.949,6.161,148.799
C06170=1179.314,97.972,-51.309,-178.951,6.159,148.799
C06171=1179.319,97.723,-51.289,-178.954,6.158,148.800
C06172=1179.324,97.474,-51.271,-178.957,6.157,148.801
C06173=1179.329,97.224,-51.253,-178.960,6.155,148.801
C06174=1179.334,96.975,-51.235,-178.962,6.154,148.802
C06175=1179.338,96.726,-51.217,-178.965,6.153,148.802
C06176=1179.343,96.476,-51.199,-178.967,6.152,148.803
C06177=1179.348,96.227,-51.181,-178.970,6.150,148.803
C06178=1179.353,95.978,-51.162,-178.973,6.150,148.804
C06179=1179.358,95.728,-51.144,-178.976,6.148,148.804
C06180=1179.363,95.479,-51.126,-178.978,6.147,148.805
C06181=1179.368,95.230,-51.108,-178.981,6.146,148.805
C06182=1179.372,94.981,-51.089,-178.983,6.145,148.806
C06183=1179.377,94.732,-51.071,-178.986,6.144,148.806
C06184=1179.382,94.482,-51.053,-178.989,6.142,148.807
C06185=1179.387,94.233,-51.035,-178.992,6.141,148.807
C06186=1179.392,93.984,-51.017,-178.994,6.140,148.808
C06187=1179.397,93.735,-50.999,-178.996,6.139,148.808
C06188=1179.401,93.485,-50.981,-179.000,6.137,148.809
C06189=1179.406,93.235,-50.964,-179.002,6.136,148.809
C06190=1179.411,92.986,-50.946,-179.005,6.135,148.810
C06191=1179.416,92.737,-50.928,-179.007,6.134,148.810
C06192=1179.421,92.488,-50.910,-179.010,6.132,148.811
C06193=1179.427,92.238,-50.891,-179.012,6.132,148.811
C06194=1179.431,91.989,-50.873,-179.015,6.130,148.812
C06195=1179.436,91.740,-50.855,-179.018,6.130,148.812
C06196=1179.441,91.491,-50.838,-179.020,6.128,148.813
C06197=1179.445,91.241,-50.820,-179.023,6.127,148.813
C06198=1179.450,90.992,-50.802,-179.026,6.126,148.814
C06199=1179.455,90.743,-50.784,-179.028,6.125,148.814
C06200=1179.460,90.493,-50.766,-179.031,6.123,148.815
C06201=1179.465,90.244,-50.748,-179.033,6.123,148.815
C06202=1179.470,89.995,-50.730,-179.036,6.121,148.816
C06203=1179.475,89.745,-50.712,-179.039,6.120,148.816
C06204=1179.480,89.496,-50.694,-179.042,6.119,148.817
C06205=1179.484,89.247,-50.677,-179.044,6.118,148.818
C06206=1179.490,88.997,-50.659,-179.047,6.116,148.818
C06207=1179.495,88.748,-50.641,-179.049,6.116,148.819
C06208=1179.499,88.499,-50.623,-179.052,6.114,148.819
C06209=1179.504,88.250,-50.605,-179.055,6.113,148.820
C06210=1179.509,88.001,-50.587,-179.057,6.112,148.820
C06211=1179.515,87.751,-50.570,-179.060,6.111,148.821
C06212=1179.518,87.501,-50.552,-179.063,6.109,148.821
C06213=1179.523,87.252,-50.534,-179.065,6.109,148.822
C06214=1179.528,87.002,-50.517,-179.068,6.107,148.822
C06215=1179.533,86.753,-50.499,-179.070,6.106,148.823
C06216=1179.538,86.504,-50.481,-179.073,6.105,148.823
C06217=1179.543,86.255,-50.463,-179.076,6.104,148.824
C06218=1179.548,86.005,-50.446,-179.079,6.103,148.824
C06219=1179.552,85.756,-50.428,-179.081,6.102,148.825
C06220=1179.557,85.507,-50.410,-179.084,6.100,148.825
C06221=1179.562,85.257,-50.393,-179.086,6.100,148.826
C06222=1179.567,85.008,-50.375,-179.089,6.098,148.826
C06223=1179.572,84.759,-50.357,-179.092,6.097,148.827
C06224=1179.578,84.509,-50.340,-179.095,6.096,148.828
C06225=1179.582,84.260,-50.323,-179.097,6.095,148.828
C06226=1179.587,84.010,-50.305,-179.100,6.093,148.828
C06227=1179.592,83.762,-50.288,-179.102,6.093,148.829
C06228=1179.597,83.513,-50.270,-179.104,6.092,148.829
C06229=1179.602,83.263,-50.253,-179.108,6.091,148.830
C06230=1179.607,83.014,-50.235,-179.110,6.090,148.831
C06231=1179.612,82.764,-50.218,-179.113,6.088,148.831
C06232=1179.617,82.515,-50.200,-179.115,6.087,148.832
C06233=1179.621,82.265,-50.183,-179.118,6.086,148.832
C06234=1179.626,82.016,-50.165,-179.120,6.085,148.833
C06235=1179.631,81.767,-50.148,-179.124,6.084,148.833
C06236=1179.636,81.517,-50.130,-179.126,6.083,148.834
C06237=1179.641,81.268,-50.113,-179.129,6.082,148.834
C06238=1179.646,81.019,-50.095,-179.131,6.081,148.835
C06239=1179.651,80.750,-50.077,-179.134,6.079,148.836
C06240=1179.657,80.482,-50.058,-179.136,6.078,148.836
C06241=1179.662,80.214,-50.039,-179.140,6.077,148.837
C06242=1179.667,79.945,-50.021,-179.143,6.076,148.837
C06243=1179.672,79.696,-50.003,-179.145,6.075,148.838
C06244=1179.677,79.446,-49.986,-179.148,6.074,148.838
C06245=1179.682,79.198,-49.969,-179.150,6.073,148.839
C06246=1179.687,78.948,-49.951,-179.153,6.072,148.839
C06247=1179.692,78.698,-49.934,-179.156,6.070,148.840
C06248=1179.696,78.449,-49.917,-179.158,6.070,148.840
C06249=1179.702,78.199,-49.899,-179.161,6.068,148.841
C06250=1179.706,77.951,-49.882,-179.164,6.068,148.842
C06251=1179.711,77.701,-49.865,-179.166,6.067,148.842
C06252=1179.717,77.452,-49.848,-179.169,6.065,148.843
C06253=1179.721,77.203,-49.830,-179.171,6.064,148.843
C06254=1179.726,76.953,-49.813,-179.174,6.063,148.844
C06255=1179.731,76.703,-49.796,-179.177,6.062,148.844
C06256=1179.736,76.454,-49.779,-179.180,6.061,148.845
C06257=1179.741,76.205,-49.761,-179.182,6.060,148.845
C06258=1179.745,75.955,-49.745,-179.185,6.059,148.846
C06259=1179.751,75.706,-49.728,-179.187,6.058,148.846
C06260=1179.755,75.457,-49.710,-179.190,6.057,148.847
C06261=1179.761,75.207,-49.693,-179.193,6.055,148.847
C06262=1179.765,74.958,-49.676,-179.195,6.055,148.848
C06263=1179.770,74.709,-49.658,-179.197,6.054,148.848
C06264=1179.776,74.460,-49.641,-179.201,6.053,148.849
C06265=1179.780,74.210,-49.625,-179.203,6.052,148.850
C06266=1179.785,73.960,-49.608,-179.206,6.050,148.850
C06267=1179.790,73.711,-49.591,-179.208,6.050,148.851
C06268=1179.795,73.462,-49.573,-179.211,6.049,148.851
C06269=1179.800,73.213,-49.557,-179.213,6.047,148.852
C06270=1179.805,72.963,-49.539,-179.216,6.047,148.852
C06271=1179.810,72.714,-49.523,-179.219,6.045,148.853
C06272=1179.815,72.464,-49.505,-179.221,6.045,148.853
C06273=1179.819,72.215,-49.488,-179.224,6.044,148.854
C06274=1179.825,71.966,-49.471,-179.227,6.042,148.855
C06275=1179.829,71.716,-49.454,-179.229,6.041,148.855
C06276=1179.835,71.467,-49.437,-179.232,6.040,148.856
C06277=1179.839,71.217,-49.421,-179.234,6.039,148.856
C06278=1179.844,70.968,-49.404,-179.237,6.039,148.857
C06279=1179.849,70.718,-49.387,-179.240,6.037,148.857
C06280=1179.854,70.469,-49.370,-179.242,6.036,148.858
C06281=1179.860,70.220,-49.353,-179.245,6.035,148.858
C06282=1179.864,69.971,-49.336,-179.248,6.034,148.859
C06283=1179.869,69.721,-49.319,-179.250,6.033,148.859
C06284=1179.873,69.472,-49.302,-179.253,6.032,148.860
C06285=1179.879,69.223,-49.286,-179.255,6.031,148.860
C06286=1179.884,68.973,-49.268,-179.258,6.031,148.861
C06287=1179.888,68.724,-49.252,-179.261,6.029,148.862
C06288=1179.893,68.474,-49.235,-179.263,6.028,148.862
C06289=1179.899,68.225,-49.218,-179.265,6.027,148.863
C06290=1179.903,67.976,-49.202,-179.269,6.026,148.863
C06291=1179.908,67.726,-49.184,-179.271,6.025,148.864
C06292=1179.913,67.477,-49.168,-179.274,6.024,148.864
C06293=1179.918,67.228,-49.151,-179.277,6.023,148.865
C06294=1179.923,66.978,-49.134,-179.279,6.023,148.865
C06295=1179.928,66.729,-49.118,-179.282,6.021,148.866
C06296=1179.933,66.480,-49.101,-179.284,6.020,148.867
C06297=1179.938,66.229,-49.085,-179.287,6.020,148.867
C06298=1179.943,65.980,-49.068,-179.289,6.018,148.868
C06299=1179.948,65.731,-49.052,-179.292,6.018,148.868
C06300=1179.953,65.481,-49.034,-179.294,6.017,148.869
C06301=1179.958,65.232,-49.018,-179.297,6.015,148.869
C06302=1179.962,64.983,-49.001,-179.300,6.014,148.870
C06303=1179.967,64.733,-48.985,-179.302,6.014,148.871
C06304=1179.973,64.484,-48.968,-179.305,6.012,148.871
C06305=1179.977,64.235,-48.951,-179.308,6.012,148.872
C06306=1179.982,63.985,-48.935,-179.310,6.010,148.872
C06307=1179.987,63.736,-48.919,-179.313,6.009,148.873
C06308=1179.992,63.486,-48.902,-179.316,6.009,148.873
C06309=1179.997,63.237,-48.885,-179.318,6.007,148.874
C06310=1180.002,62.988,-48.869,-179.321,6.007,148.874
C06311=1180.006,62.738,-48.852,-179.323,6.006,148.875
C06312=1180.012,62.489,-48.836,-179.326,6.005,148.876
C06313=1180.017,62.239,-48.819,-179.328,6.004,148.876
C06314=1180.022,61.990,-48.803,-179.331,6.003,148.877
C06315=1180.027,61.741,-48.786,-179.334,6.001,148.877
C06316=1180.031,61.491,-48.770,-179.336,6.001,148.878
C06317=1180.037,61.242,-48.753,-179.339,6.000,148.878
C06318=1180.042,60.992,-48.737,-179.341,5.999,148.879
C06319=1180.047,60.743,-48.720,-179.344,5.998,148.880
C06320=1180.051,60.493,-48.704,-179.347,5.997,148.880
C06321=1180.057,60.244,-48.688,-179.349,5.997,148.881
C06322=1180.062,59.995,-48.671,-179.352,5.995,148.881
C06323=1180.067,59.745,-48.655,-179.355,5.995,148.882
C06324=1180.072,59.496,-48.639,-179.357,5.994,148.882
C06325=1180.076,59.246,-48.622,-179.360,5.992,148.883
C06326=1180.082,58.997,-48.606,-179.363,5.992,148.883
C06327=1180.086,58.747,-48.590,-179.365,5.991,148.884
C06328=1180.091,58.499,-48.573,-179.368,5.990,148.885
C06329=1180.096,58.249,-48.557,-179.370,5.989,148.885
C06330=1180.102,57.999,-48.540,-179.373,5.988,148.886
C06331=1180.106,57.750,-48.524,-179.375,5.986,148.886
C06332=1180.112,57.501,-48.508,-179.378,5.986,148.887
C06333=1180.116,57.251,-48.492,-179.381,5.985,148.887
C06334=1180.121,57.002,-48.476,-179.383,5.985,148.888
C06335=1180.126,56.752,-48.459,-179.386,5.983,148.889
C06336=1180.131,56.503,-48.444,-179.388,5.982,148.889
C06337=1180.136,56.253,-48.427,-179.391,5.982,148.890
C06338=1180.141,56.005,-48.411,-179.394,5.980,148.890
C06339=1180.146,55.754,-48.395,-179.396,5.980,148.891
C06340=1180.151,55.506,-48.378,-179.398,5.979,148.891
C06341=1180.155,55.256,-48.362,-179.402,5.977,148.892
C06342=1180.161,55.007,-48.346,-179.404,5.977,148.893
C06343=1180.166,54.737,-48.328,-179.406,5.976,148.893
C06344=1180.172,54.469,-48.311,-179.410,5.975,148.894
C06345=1180.177,54.201,-48.293,-179.412,5.974,148.894
C06346=1180.183,53.932,-48.276,-179.415,5.973,148.895
C06347=1180.187,53.682,-48.260,-179.418,5.972,148.895
C06348=1180.193,53.434,-48.244,-179.420,5.971,148.896
C06349=1180.197,53.183,-48.228,-179.422,5.971,148.897
C06350=1180.202,52.935,-48.212,-179.426,5.969,148.897
C06351=1180.207,52.685,-48.196,-179.428,5.969,148.898
C06352=1180.213,52.435,-48.180,-179.430,5.968,148.898
C06353=1180.217,52.186,-48.164,-179.434,5.967,148.899
C06354=1180.222,51.936,-48.148,-179.436,5.966,148.899
C06355=1180.227,51.687,-48.132,-179.438,5.965,148.900
C06356=1180.232,51.438,-48.116,-179.441,5.965,148.901
C06357=1180.237,51.188,-48.101,-179.444,5.963,148.901
C06358=1180.241,50.939,-48.084,-179.446,5.962,148.902
C06359=1180.247,50.689,-48.069,-179.449,5.962,148.902
C06360=1180.252,50.440,-48.053,-179.451,5.961,148.903
C06361=1180.257,50.191,-48.036,-179.454,5.960,148.904
C06362=1180.262,49.941,-48.021,-179.457,5.959,148.904
C06363=1180.267,49.691,-48.005,-179.459,5.958,148.905
C06364=1180.272,49.442,-47.989,-179.461,5.957,148.905
C06365=1180.277,49.193,-47.973,-179.465,5.956,148.906
C06366=1180.281,48.943,-47.958,-179.467,5.955,148.906
C06367=1180.286,48.694,-47.941,-179.469,5.955,148.907
C06368=1180.291,48.444,-47.925,-179.472,5.954,148.908
C06369=1180.297,48.195,-47.910,-179.475,5.953,148.908
C06370=1180.302,47.945,-47.894,-179.477,5.952,148.909
C06371=1180.306,47.696,-47.877,-179.480,5.951,148.909
C06372=1180.312,47.446,-47.862,-179.482,5.951,148.910
C06373=1180.317,47.197,-47.847,-179.485,5.949,148.910
C06374=1180.321,46.947,-47.831,-179.488,5.948,148.911
C06375=1180.326,46.698,-47.815,-179.490,5.948,148.912
C06376=1180.332,46.449,-47.799,-179.492,5.947,148.912
C06377=1180.337,46.199,-47.783,-179.496,5.946,148.913
C06378=1180.342,45.950,-47.768,-179.498,5.945,148.913
C06379=1180.347,45.700,-47.753,-179.500,5.944,148.914
C06380=1180.351,45.451,-47.736,-179.503,5.944,148.915
C06381=1180.356,45.202,-47.720,-179.506,5.942,148.915
C06382=1180.362,44.952,-47.705,-179.508,5.942,148.916
C06383=1180.366,44.702,-47.689,-179.511,5.941,148.916
C06384=1180.371,44.453,-47.674,-179.513,5.940,148.917
C06385=1180.377,44.204,-47.658,-179.516,5.940,148.917
C06386=1180.382,43.954,-47.643,-179.519,5.938,148.918
C06387=1180.386,43.704,-47.627,-179.521,5.938,148.919
C06388=1180.391,43.456,-47.611,-179.524,5.937,148.919
C06389=1180.397,43.206,-47.595,-179.526,5.936,148.920
C06390=1180.401,42.956,-47.579,-179.529,5.935,148.920
C06391=1180.406,42.707,-47.564,-179.532,5.934,148.921
C06392=1180.411,42.458,-47.549,-179.534,5.934,148.921
C06393=1180.417,42.208,-47.533,-179.537,5.933,148.922
C06394=1180.422,41.958,-47.517,-179.539,5.932,148.923
C06395=1180.426,41.709,-47.502,-179.542,5.931,148.923
C06396=1180.432,41.460,-47.487,-179.545,5.930,148.924
C06397=1180.437,41.210,-47.471,-179.547,5.929,148.924
C06398=1180.441,40.960,-47.456,-179.550,5.929,148.925
C06399=1180.446,40.711,-47.440,-179.552,5.928,148.926
C06400=1180.452,40.462,-47.425,-179.555,5.927,148.926
C06401=1180.456,40.213,-47.410,-179.558,5.926,148.927
C06402=1180.461,39.962,-47.394,-179.560,5.925,148.927
C06403=1180.467,39.713,-47.378,-179.562,5.925,148.928
C06404=1180.471,39.464,-47.363,-179.565,5.924,148.929
C06405=1180.477,39.215,-47.347,-179.568,5.923,148.929
C06406=1180.482,38.965,-47.332,-179.570,5.922,148.930
C06407=1180.486,38.715,-47.316,-179.573,5.922,148.930
C06408=1180.491,38.466,-47.301,-179.575,5.921,148.931
C06409=1180.496,38.217,-47.286,-179.578,5.920,148.931
C06410=1180.502,37.967,-47.271,-179.581,5.919,148.932
C06411=1180.507,37.717,-47.255,-179.583,5.918,148.933
C06412=1180.511,37.468,-47.240,-179.586,5.918,148.933
C06413=1180.517,37.218,-47.224,-179.588,5.917,148.934
C06414=1180.521,36.969,-47.209,-179.591,5.916,148.934
C06415=1180.527,36.720,-47.194,-179.593,5.916,148.935
C06416=1180.532,36.470,-47.178,-179.596,5.914,148.936
C06417=1180.537,36.221,-47.164,-179.599,5.914,148.936
C06418=1180.542,35.970,-47.148,-179.601,5.913,148.937
C06419=1180.546,35.721,-47.133,-179.603,5.912,148.937
C06420=1180.552,35.472,-47.117,-179.606,5.912,148.938
C06421=1180.556,35.223,-47.103,-179.608,5.911,148.938
C06422=1180.562,34.974,-47.087,-179.611,5.910,148.939
C06423=1180.567,34.724,-47.073,-179.614,5.909,148.940
C06424=1180.572,34.474,-47.057,-179.616,5.908,148.940
C06425=1180.576,34.225,-47.042,-179.619,5.908,148.941
C06426=1180.582,33.975,-47.026,-179.621,5.907,148.941
C06427=1180.587,33.725,-47.012,-179.624,5.906,148.942
C06428=1180.592,33.476,-46.996,-179.627,5.905,148.943
C06429=1180.597,33.227,-46.981,-179.629,5.904,148.943
C06430=1180.602,32.978,-46.966,-179.632,5.904,148.944
C06431=1180.607,32.728,-46.951,-179.634,5.903,148.945
C06432=1180.612,32.478,-46.936,-179.637,5.902,148.945
C06433=1180.616,32.229,-46.920,-179.639,5.902,148.946
C06434=1180.622,31.979,-46.906,-179.642,5.901,148.946
C06435=1180.627,31.730,-46.891,-179.645,5.900,148.947
C06436=1180.632,31.480,-46.875,-179.647,5.899,148.947
C06437=1180.637,31.230,-46.861,-179.650,5.899,148.948
C06438=1180.642,30.981,-46.846,-179.652,5.898,148.949
C06439=1180.647,30.732,-46.830,-179.655,5.897,148.949
C06440=1180.652,30.482,-46.816,-179.657,5.896,148.950
C06441=1180.657,30.233,-46.800,-179.660,5.895,148.950
C06442=1180.662,29.984,-46.785,-179.663,5.895,148.951
C06443=1180.668,29.734,-46.770,-179.665,5.894,148.952
C06444=1180.672,29.485,-46.755,-179.668,5.893,148.952
C06445=1180.677,29.235,-46.741,-179.670,5.893,148.953
C06446=1180.683,28.986,-46.726,-179.672,5.892,148.953
C06447=1180.688,28.717,-46.710,-179.676,5.891,148.954
C06448=1180.694,28.448,-46.694,-179.678,5.890,148.955
C06449=1180.699,28.179,-46.678,-179.681,5.890,148.955
C06450=1180.704,27.910,-46.661,-179.684,5.889,148.956
C06451=1180.709,27.661,-46.647,-179.686,5.887,148.956
C06452=1180.714,27.412,-46.632,-179.689,5.887,148.957
C06453=1180.720,27.162,-46.617,-179.692,5.886,148.958
C06454=1180.724,26.912,-46.602,-179.694,5.886,148.958
C06455=1180.729,26.663,-46.587,-179.696,5.885,148.959
C06456=1180.735,26.413,-46.572,-179.699,5.885,148.960
C06457=1180.739,26.163,-46.557,-179.701,5.884,148.960
C06458=1180.744,25.915,-46.543,-179.704,5.883,148.961
C06459=1180.749,25.665,-46.528,-179.707,5.882,148.961
C06460=1180.755,25.415,-46.513,-179.709,5.881,148.962
C06461=1180.760,25.166,-46.498,-179.712,5.881,148.963
C06462=1180.765,24.916,-46.484,-179.714,5.880,148.963
C06463=1180.770,24.667,-46.469,-179.717,5.879,148.964
C06464=1180.775,24.417,-46.454,-179.719,5.879,148.964
C06465=1180.780,24.168,-46.439,-179.722,5.878,148.965
C06466=1180.785,23.918,-46.425,-179.724,5.877,148.966
C06467=1180.790,23.669,-46.409,-179.727,5.877,148.966
C06468=1180.795,23.419,-46.395,-179.730,5.876,148.967
C06469=1180.800,23.169,-46.381,-179.732,5.875,148.967
C06470=1180.805,22.920,-46.366,-179.735,5.874,148.968
C06471=1180.810,22.670,-46.351,-179.737,5.874,148.969
C06472=1180.815,22.420,-46.337,-179.740,5.873,148.969
C06473=1180.820,22.171,-46.322,-179.742,5.872,148.970
C06474=1180.825,21.922,-46.307,-179.745,5.872,148.971
C06475=1180.830,21.672,-46.293,-179.747,5.871,148.971
C06476=1180.835,21.423,-46.278,-179.750,5.871,148.972
C06477=1180.840,21.173,-46.263,-179.752,5.870,148.972
C06478=1180.845,20.923,-46.249,-179.755,5.868,148.973
C06479=1180.850,20.674,-46.234,-179.758,5.868,148.973
C06480=1180.855,20.424,-46.220,-179.760,5.868,148.974
C06481=1180.861,20.175,-46.205,-179.763,5.867,148.975
C06482=1180.866,19.926,-46.190,-179.765,5.866,148.975
C06483=1180.871,19.676,-46.176,-179.768,5.866,148.976
C06484=1180.875,19.426,-46.162,-179.770,5.865,148.976
C06485=1180.880,19.177,-46.147,-179.773,5.864,148.977
C06486=1180.885,18.928,-46.132,-179.775,5.864,148.978
C06487=1180.890,18.678,-46.118,-179.777,5.863,148.978
C06488=1180.896,18.428,-46.103,-179.780,5.863,148.979
C06489=1180.901,18.178,-46.089,-179.783,5.862,148.980
C06490=1180.906,17.929,-46.075,-179.786,5.860,148.980
C06491=1180.911,17.680,-46.060,-179.788,5.860,148.981
C06492=1180.916,17.430,-46.046,-179.791,5.859,148.981
C06493=1180.921,17.181,-46.032,-179.793,5.859,148.982
C06494=1180.926,16.931,-46.017,-179.796,5.858,148.983
C06495=1180.931,16.681,-46.003,-179.798,5.858,148.983
C06496=1180.936,16.432,-45.989,-179.800,5.857,148.984
C06497=1180.941,16.183,-45.974,-179.803,5.856,148.984
C06498=1180.947,15.933,-45.959,-179.806,5.856,148.985
C06499=1180.952,15.683,-45.945,-179.808,5.855,148.985
C06500=1180.957,15.434,-45.931,-179.811,5.854,148.986
C06501=1180.961,15.184,-45.916,-179.813,5.854,148.987
C06502=1180.966,14.934,-45.902,-179.815,5.853,148.987
C06503=1180.972,14.685,-45.888,-179.818,5.853,148.988
C06504=1180.977,14.436,-45.874,-179.821,5.852,148.989
C06505=1180.982,14.186,-45.860,-179.823,5.851,148.989
C06506=1180.987,13.937,-45.845,-179.826,5.850,148.990
C06507=1180.991,13.687,-45.830,-179.829,5.849,148.991
C06508=1180.997,13.438,-45.816,-179.831,5.849,148.991
C06509=1181.002,13.188,-45.802,-179.834,5.848,148.992
C06510=1181.007,12.939,-45.788,-179.836,5.848,148.992
C06511=1181.012,12.689,-45.774,-179.838,5.847,148.993
C06512=1181.017,12.439,-45.759,-179.841,5.846,148.993
C06513=1181.022,12.190,-45.745,-179.844,5.846,148.994
C06514=1181.027,11.941,-45.731,-179.846,5.845,148.995
C06515=1181.032,11.691,-45.717,-179.848,5.845,148.995
C06516=1181.037,11.441,-45.703,-179.851,5.844,148.996
C06517=1181.043,11.192,-45.689,-179.854,5.844,148.997
C06518=1181.048,10.942,-45.674,-179.856,5.843,148.997
C06519=1181.053,10.693,-45.660,-179.859,5.842,148.998
C06520=1181.058,10.443,-45.646,-179.861,5.842,148.998
C06521=1181.063,10.194,-45.633,-179.863,5.841,148.999
C06522=1181.068,9.944,-45.619,-179.866,5.840,149.000
C06523=1181.073,9.694,-45.605,-179.869,5.840,149.000
C06524=1181.078,9.445,-45.590,-179.871,5.839,149.001
C06525=1181.083,9.196,-45.577,-179.874,5.839,149.001
C06526=1181.088,8.946,-45.562,-179.876,5.838,149.002
C06527=1181.093,8.696,-45.548,-179.878,5.837,149.003
C06528=1181.098,8.446,-45.534,-179.881,5.837,149.003
C06529=1181.104,8.197,-45.520,-179.884,5.836,149.004
C06530=1181.109,7.948,-45.505,-179.886,5.835,149.004
C06531=1181.113,7.698,-45.493,-179.888,5.835,149.005
C06532=1181.119,7.449,-45.479,-179.891,5.835,149.006
C06533=1181.124,7.199,-45.464,-179.893,5.834,149.006
C06534=1181.129,6.949,-45.450,-179.896,5.833,149.007
C06535=1181.134,6.699,-45.436,-179.899,5.833,149.008
C06536=1181.139,6.450,-45.422,-179.901,5.832,149.008
C06537=1181.144,6.200,-45.408,-179.903,5.831,149.009
C06538=1181.149,5.951,-45.395,-179.906,5.831,149.009
C06539=1181.154,5.702,-45.381,-179.909,5.830,149.010
C06540=1181.159,5.452,-45.366,-179.911,5.829,149.011
C06541=1181.164,5.202,-45.352,-179.914,5.828,149.011
C06542=1181.170,4.953,-45.339,-179.917,5.828,149.012
C06543=1181.174,4.703,-45.325,-179.919,5.827,149.012
C06544=1181.179,4.454,-45.311,-179.922,5.827,149.013
C06545=1181.185,4.205,-45.297,-179.924,5.826,149.014
C06546=1181.190,3.954,-45.284,-179.926,5.825,149.014
C06547=1181.195,3.705,-45.269,-179.929,5.825,149.015
C06548=1181.200,3.456,-45.256,-179.932,5.824,149.016
C06549=1181.205,3.206,-45.242,-179.934,5.824,149.016
C06550=1181.210,2.956,-45.228,-179.937,5.823,149.017
C06551=1181.216,2.687,-45.213,-179.939,5.822,149.017
C06552=1181.221,2.418,-45.198,-179.942,5.822,149.018
C06553=1181.227,2.148,-45.183,-179.945,5.822,149.019
C06554=1181.232,1.879,-45.169,-179.947,5.821,149.020
C06555=1181.237,1.630,-45.155,-179.950,5.821,149.020
C06556=1181.242,1.380,-45.141,-179.952,5.820,149.021
C06557=1181.247,1.130,-45.127,-179.955,5.819,149.021
C06558=1181.252,0.881,-45.114,-179.957,5.819,149.022
C06559=1181.257,0.631,-45.100,-179.959,5.818,149.023
C06560=1181.263,0.382,-45.087,-179.962,5.817,149.023
C06561=1181.267,0.133,-45.073,-179.965,5.817,149.024
C06562=1181.273,-0.117,-45.060,-179.967,5.816,149.024
C06563=1181.278,-0.367,-45.045,-179.970,5.816,149.025
C06564=1181.283,-0.617,-45.032,-179.972,5.815,149.026
C06565=1181.288,-0.866,-45.019,-179.975,5.815,149.026
C06566=1181.293,-1.115,-45.004,-179.977,5.814,149.027
C06567=1181.299,-1.365,-44.991,-179.980,5.813,149.028
C06568=1181.303,-1.614,-44.977,-179.982,5.813,149.028
C06569=1181.308,-1.865,-44.964,-179.985,5.812,149.029
C06570=1181.314,-2.114,-44.950,-179.987,5.812,149.029
C06571=1181.318,-2.364,-44.937,-179.990,5.811,149.030
C06572=1181.324,-2.613,-44.923,-179.992,5.810,149.031
C06573=1181.328,-2.863,-44.910,-179.995,5.810,149.031
C06574=1181.334,-3.112,-44.896,-179.997,5.809,149.032
C06575=1181.339,-3.362,-44.883,-180.000,5.809,149.032
C06576=1181.344,-3.611,-44.869,179.998,5.808,149.033
C06577=1181.349,-3.861,-44.856,179.996,5.808,149.034
C06578=1181.354,-4.110,-44.842,179.993,5.808,149.035
C06579=1181.359,-4.360,-44.829,179.991,5.807,149.035
C06580=1181.365,-4.609,-44.815,179.988,5.807,149.036
C06581=1181.370,-4.859,-44.802,179.986,5.806,149.036
C06582=1181.375,-5.108,-44.788,179.983,5.805,149.037
C06583=1181.380,-5.358,-44.775,179.981,5.805,149.037
C06584=1181.385,-5.608,-44.762,179.978,5.804,149.038
C06585=1181.390,-5.857,-44.748,179.976,5.804,149.039
C06586=1181.396,-6.107,-44.735,179.973,5.803,149.039
C06587=1181.400,-6.357,-44.721,179.971,5.803,149.040
C06588=1181.406,-6.606,-44.708,179.968,5.802,149.041
C06589=1181.411,-6.856,-44.695,179.966,5.801,149.041
C06590=1181.416,-7.105,-44.681,179.963,5.801,149.042
C06591=1181.421,-7.355,-44.668,179.961,5.800,149.043
C06592=1181.426,-7.605,-44.655,179.958,5.800,149.043
C06593=1181.431,-7.854,-44.641,179.956,5.799,149.044
C06594=1181.436,-8.104,-44.628,179.953,5.799,149.044
C06595=1181.441,-8.354,-44.615,179.950,5.798,149.045
C06596=1181.446,-8.603,-44.601,179.949,5.798,149.046
C06597=1181.452,-8.853,-44.588,179.946,5.798,149.046
C06598=1181.457,-9.102,-44.575,179.943,5.797,149.047
C06599=1181.462,-9.352,-44.561,179.941,5.796,149.047
C06600=1181.467,-9.601,-44.548,179.939,5.796,149.048
C06601=1181.472,-9.852,-44.535,179.936,5.795,149.049
C06602=1181.477,-10.100,-44.521,179.934,5.795,149.049
C06603=1181.482,-10.350,-44.509,179.931,5.794,149.050
C06604=1181.487,-10.600,-44.495,179.928,5.794,149.051
C06605=1181.492,-10.849,-44.483,179.926,5.793,149.051
C06606=1181.497,-11.099,-44.468,179.924,5.792,149.052
C06607=1181.502,-11.348,-44.456,179.921,5.792,149.053
C06608=1181.508,-11.599,-44.442,179.918,5.791,149.053
C06609=1181.513,-11.848,-44.430,179.916,5.791,149.054
C06610=1181.518,-12.097,-44.416,179.914,5.791,149.054
C06611=1181.523,-12.347,-44.403,179.911,5.790,149.055
C06612=1181.528,-12.596,-44.390,179.909,5.790,149.056
C06613=1181.533,-12.847,-44.377,179.907,5.789,149.056
C06614=1181.538,-13.096,-44.364,179.904,5.789,149.057
C06615=1181.543,-13.345,-44.351,179.901,5.788,149.058
C06616=1181.548,-13.595,-44.337,179.899,5.787,149.058
C06617=1181.554,-13.844,-44.324,179.896,5.787,149.059
C06618=1181.559,-14.095,-44.311,179.894,5.787,149.059
C06619=1181.564,-14.344,-44.298,179.892,5.786,149.060
C06620=1181.569,-14.593,-44.286,179.889,5.785,149.061
C06621=1181.574,-14.844,-44.272,179.887,5.786,149.061
C06622=1181.579,-15.093,-44.260,179.884,5.785,149.062
C06623=1181.584,-15.342,-44.246,179.882,5.784,149.062
C06624=1181.590,-15.592,-44.233,179.879,5.784,149.063
C06625=1181.595,-15.841,-44.220,179.877,5.783,149.064
C06626=1181.600,-16.091,-44.207,179.875,5.783,149.064
C06627=1181.605,-16.341,-44.194,179.872,5.782,149.065
C06628=1181.610,-16.590,-44.181,179.869,5.782,149.066
C06629=1181.615,-16.840,-44.169,179.867,5.781,149.066
C06630=1181.621,-17.090,-44.155,179.864,5.780,149.067
C06631=1181.626,-17.339,-44.143,179.862,5.781,149.068
C06632=1181.631,-17.589,-44.130,179.860,5.780,149.068
C06633=1181.635,-17.839,-44.117,179.858,5.779,149.069
C06634=1181.641,-18.088,-44.104,179.855,5.779,149.069
C06635=1181.646,-18.338,-44.091,179.852,5.778,149.070
C06636=1181.651,-18.588,-44.078,179.850,5.778,149.071
C06637=1181.657,-18.837,-44.065,179.847,5.777,149.071
C06638=1181.662,-19.087,-44.052,179.845,5.777,149.072
C06639=1181.666,-19.337,-44.039,179.842,5.776,149.073
C06640=1181.671,-19.586,-44.027,179.840,5.776,149.073
C06641=1181.677,-19.835,-44.014,179.838,5.776,149.074
C06642=1181.682,-20.085,-44.001,179.835,5.775,149.075
C06643=1181.687,-20.335,-43.988,179.833,5.774,149.075
C06644=1181.692,-20.584,-43.975,179.830,5.774,149.076
C06645=1181.697,-20.833,-43.963,179.828,5.774,149.076
C06646=1181.703,-21.083,-43.950,179.825,5.773,149.077
C06647=1181.708,-21.333,-43.937,179.823,5.772,149.078
C06648=1181.713,-21.582,-43.924,179.821,5.773,149.078
C06649=1181.718,-21.832,-43.912,179.818,5.772,149.079
C06650=1181.723,-22.083,-43.899,179.816,5.771,149.079
C06651=1181.729,-22.332,-43.886,179.813,5.771,149.080
C06652=1181.734,-22.581,-43.873,179.811,5.770,149.081
C06653=1181.739,-22.831,-43.861,179.808,5.770,149.081
C06654=1181.744,-23.080,-43.848,179.806,5.769,149.082
C06655=1181.750,-23.350,-43.834,179.803,5.769,149.083
C06656=1181.755,-23.620,-43.820,179.800,5.768,149.083
C06657=1181.761,-23.889,-43.808,179.798,5.768,149.084
C06658=1181.766,-24.159,-43.793,179.795,5.767,149.085
C06659=1181.771,-24.409,-43.781,179.793,5.768,149.085
C06660=1181.776,-24.659,-43.768,179.791,5.767,149.086
C06661=1181.781,-24.908,-43.755,179.788,5.766,149.087
C06662=1181.786,-25.158,-43.743,179.786,5.766,149.087
C06663=1181.792,-25.407,-43.731,179.783,5.765,149.088
C06664=1181.797,-25.657,-43.718,179.781,5.765,149.088
C06665=1181.802,-25.907,-43.705,179.778,5.764,149.089
C06666=1181.807,-26.156,-43.692,179.776,5.764,149.090
C06667=1181.813,-26.406,-43.680,179.774,5.764,149.090
C06668=1181.818,-26.656,-43.668,179.771,5.763,149.091
C06669=1181.823,-26.905,-43.655,179.768,5.763,149.092
C06670=1181.827,-27.155,-43.642,179.766,5.762,149.092
C06671=1181.833,-27.405,-43.630,179.764,5.762,149.093
C06672=1181.838,-27.654,-43.617,179.761,5.761,149.094
C06673=1181.843,-27.903,-43.605,179.759,5.761,149.094
C06674=1181.848,-28.153,-43.593,179.757,5.761,149.095
C06675=1181.854,-28.403,-43.580,179.754,5.760,149.095
C06676=1181.858,-28.653,-43.567,179.751,5.760,149.096
C06677=1181.863,-28.902,-43.555,179.749,5.759,149.097
C06678=1181.869,-29.152,-43.543,179.747,5.759,149.097
C06679=1181.874,-29.401,-43.530,179.745,5.759,149.098
C06680=1181.880,-29.651,-43.517,179.742,5.758,149.098
C06681=1181.885,-29.901,-43.505,179.740,5.758,149.099
C06682=1181.890,-30.151,-43.492,179.737,5.757,149.100
C06683=1181.895,-30.401,-43.480,179.735,5.756,149.100
C06684=1181.900,-30.650,-43.468,179.732,5.756,149.101
C06685=1181.905,-30.899,-43.455,179.730,5.756,149.102
C06686=1181.911,-31.149,-43.443,179.727,5.756,149.102
C06687=1181.915,-31.398,-43.431,179.725,5.755,149.103
C06688=1181.920,-31.648,-43.419,179.723,5.755,149.104
C06689=1181.926,-31.898,-43.407,179.720,5.754,149.104
C06690=1181.931,-32.147,-43.394,179.718,5.753,149.105
C06691=1181.936,-32.398,-43.382,179.716,5.754,149.105
C06692=1181.941,-32.647,-43.369,179.713,5.753,149.106
C06693=1181.946,-32.897,-43.357,179.711,5.752,149.107
C06694=1181.951,-33.146,-43.345,179.708,5.752,149.107
C06695=1181.957,-33.396,-43.333,179.706,5.751,149.108
C06696=1181.962,-33.645,-43.320,179.703,5.752,149.109
C06697=1181.967,-33.895,-43.308,179.701,5.751,149.109
C06698=1181.972,-34.145,-43.296,179.699,5.751,149.110
C06699=1181.977,-34.394,-43.283,179.696,5.750,149.111
C06700=1181.983,-34.644,-43.271,179.694,5.749,149.111
C06701=1181.988,-34.893,-43.259,179.692,5.750,149.112
C06702=1181.993,-35.143,-43.247,179.689,5.749,149.112
C06703=1181.998,-35.393,-43.234,179.686,5.749,149.113
C06704=1182.003,-35.643,-43.223,179.684,5.748,149.114
C06705=1182.008,-35.893,-43.211,179.682,5.747,149.114
C06706=1182.013,-36.142,-43.198,179.679,5.748,149.115
C06707=1182.019,-36.392,-43.186,179.677,5.747,149.116
C06708=1182.024,-36.641,-43.174,179.675,5.747,149.116
C06709=1182.029,-36.891,-43.162,179.672,5.746,149.117
C06710=1182.034,-37.141,-43.149,179.670,5.745,149.117
C06711=1182.040,-37.391,-43.137,179.667,5.745,149.118
C06712=1182.044,-37.640,-43.126,179.665,5.745,149.119
C06713=1182.050,-37.889,-43.113,179.662,5.745,149.119
C06714=1182.055,-38.139,-43.102,179.660,5.744,149.120
C06715=1182.060,-38.389,-43.089,179.658,5.744,149.121
C06716=1182.066,-38.639,-43.077,179.655,5.744,149.121
C06717=1182.071,-38.889,-43.065,179.653,5.743,149.122
C06718=1182.075,-39.138,-43.053,179.651,5.743,149.123
C06719=1182.081,-39.388,-43.041,179.648,5.742,149.123
C06720=1182.086,-39.637,-43.029,179.646,5.741,149.124
C06721=1182.091,-39.887,-43.017,179.644,5.742,149.124
C06722=1182.097,-40.137,-43.005,179.641,5.741,149.125
C06723=1182.101,-40.386,-42.993,179.639,5.740,149.126
C06724=1182.107,-40.636,-42.981,179.636,5.740,149.126
C06725=1182.112,-40.886,-42.969,179.633,5.740,149.127
C06726=1182.117,-41.136,-42.957,179.631,5.740,149.128
C06727=1182.122,-41.385,-42.945,179.629,5.739,149.128
C06728=1182.127,-41.634,-42.933,179.627,5.739,149.129
C06729=1182.133,-41.884,-42.921,179.624,5.738,149.130
C06730=1182.138,-42.134,-42.909,179.622,5.738,149.130
C06731=1182.143,-42.383,-42.898,179.620,5.738,149.131
C06732=1182.148,-42.633,-42.886,179.617,5.737,149.131
C06733=1182.153,-42.883,-42.874,179.615,5.737,149.132
C06734=1182.158,-43.133,-42.861,179.612,5.736,149.133
C06735=1182.164,-43.381,-42.850,179.610,5.736,149.133
C06736=1182.169,-43.631,-42.838,179.607,5.736,149.134
C06737=1182.175,-43.881,-42.827,179.605,5.735,149.134
C06738=1182.180,-44.131,-42.814,179.603,5.735,149.135
C06739=1182.184,-44.380,-42.803,179.600,5.735,149.136
C06740=1182.190,-44.630,-42.791,179.598,5.734,149.136
C06741=1182.195,-44.880,-42.779,179.596,5.734,149.137
C06742=1182.200,-45.130,-42.768,179.593,5.733,149.138
C06743=1182.205,-45.379,-42.755,179.591,5.733,149.138
C06744=1182.211,-45.629,-42.743,179.589,5.733,149.139
C06745=1182.215,-45.879,-42.732,179.586,5.733,149.140
C06746=1182.221,-46.129,-42.720,179.584,5.732,149.140
C06747=1182.226,-46.379,-42.708,179.582,5.732,149.141
C06748=1182.231,-46.627,-42.697,179.579,5.732,149.142
C06749=1182.237,-46.877,-42.685,179.576,5.731,149.142
C06750=1182.242,-47.127,-42.673,179.574,5.730,149.143
C06751=1182.247,-47.376,-42.661,179.572,5.730,149.143
C06752=1182.252,-47.626,-42.649,179.570,5.730,149.144
C06753=1182.258,-47.876,-42.638,179.567,5.730,149.145
C06754=1182.262,-48.126,-42.626,179.565,5.729,149.145
C06755=1182.268,-48.376,-42.614,179.562,5.729,149.146
C06756=1182.273,-48.625,-42.603,179.560,5.729,149.146
C06757=1182.278,-48.875,-42.592,179.558,5.728,149.147
C06758=1182.284,-49.125,-42.580,179.555,5.728,149.148
C06759=1182.289,-49.395,-42.567,179.552,5.727,149.149
C06760=1182.295,-49.665,-42.554,179.550,5.727,149.149
C06761=1182.301,-49.936,-42.542,179.548,5.727,149.150
C06762=1182.306,-50.206,-42.529,179.546,5.727,149.150
C06763=1182.311,-50.456,-42.518,179.543,5.726,149.151
C06764=1182.317,-50.705,-42.506,179.540,5.726,149.152
C06765=1182.321,-50.954,-42.495,179.538,5.725,149.152
C06766=1182.327,-51.204,-42.483,179.536,5.725,149.153
C06767=1182.331,-51.454,-42.472,179.533,5.725,149.154
C06768=1182.337,-51.704,-42.460,179.531,5.724,149.154
C06769=1182.342,-51.954,-42.448,179.529,5.724,149.155
C06770=1182.348,-52.203,-42.437,179.526,5.724,149.156
C06771=1182.352,-52.452,-42.426,179.524,5.724,149.156
C06772=1182.358,-52.702,-42.414,179.521,5.723,149.157
C06773=1182.363,-52.952,-42.402,179.519,5.723,149.157
C06774=1182.368,-53.202,-42.391,179.517,5.723,149.158
C06775=1182.374,-53.451,-42.379,179.515,5.722,149.159
C06776=1182.379,-53.701,-42.368,179.512,5.721,149.159
C06777=1182.384,-53.951,-42.356,179.510,5.722,149.160
C06778=1182.389,-54.201,-42.345,179.508,5.721,149.161
C06779=1182.394,-54.451,-42.334,179.505,5.721,149.161
C06780=1182.400,-54.700,-42.323,179.503,5.721,149.162
C06781=1182.404,-54.949,-42.311,179.501,5.720,149.162
C06782=1182.410,-55.199,-42.299,179.498,5.720,149.163
C06783=1182.415,-55.449,-42.288,179.495,5.719,149.164
C06784=1182.420,-55.699,-42.276,179.494,5.719,149.164
C06785=1182.425,-55.948,-42.265,179.491,5.719,149.165
C06786=1182.431,-56.198,-42.253,179.488,5.718,149.166
C06787=1182.436,-56.448,-42.243,179.486,5.718,149.166
C06788=1182.441,-56.698,-42.231,179.484,5.718,149.167
C06789=1182.446,-56.947,-42.220,179.481,5.718,149.168
C06790=1182.451,-57.197,-42.209,179.479,5.717,149.168
C06791=1182.457,-57.446,-42.197,179.477,5.717,149.169
C06792=1182.461,-57.696,-42.186,179.475,5.717,149.170
C06793=1182.468,-57.946,-42.175,179.472,5.716,149.170
C06794=1182.472,-58.196,-42.163,179.470,5.716,149.171
C06795=1182.477,-58.445,-42.152,179.468,5.716,149.171
C06796=1182.482,-58.695,-42.140,179.465,5.715,149.172
C06797=1182.488,-58.944,-42.129,179.463,5.715,149.173
C06798=1182.493,-59.195,-42.118,179.461,5.715,149.173
C06799=1182.498,-59.444,-42.107,179.458,5.715,149.174
C06800=1182.503,-59.693,-42.096,179.456,5.714,149.174
C06801=1182.509,-59.943,-42.084,179.454,5.714,149.175
C06802=1182.514,-60.193,-42.073,179.451,5.714,149.176
C06803=1182.519,-60.443,-42.062,179.449,5.713,149.176
C06804=1182.525,-60.692,-42.051,179.446,5.712,149.177
C06805=1182.529,-60.942,-42.039,179.444,5.713,149.178
C06806=1182.534,-61.192,-42.029,179.442,5.712,149.178
C06807=1182.540,-61.441,-42.017,179.439,5.712,149.179
C06808=1182.545,-61.691,-42.006,179.437,5.712,149.180
C06809=1182.550,-61.941,-41.995,179.435,5.711,149.180
C06810=1182.556,-62.190,-41.984,179.432,5.711,149.181
C06811=1182.561,-62.440,-41.973,179.430,5.711,149.182
C06812=1182.566,-62.690,-41.962,179.428,5.710,149.182
C06813=1182.572,-62.940,-41.951,179.425,5.710,149.183
C06814=1182.576,-63.189,-41.939,179.423,5.710,149.183
C06815=1182.581,-63.439,-41.929,179.421,5.709,149.184
C06816=1182.587,-63.689,-41.917,179.419,5.709,149.185
C06817=1182.592,-63.938,-41.906,179.416,5.709,149.185
C06818=1182.597,-64.188,-41.895,179.414,5.709,149.186
C06819=1182.602,-64.437,-41.884,179.412,5.708,149.186
C06820=1182.608,-64.688,-41.873,179.409,5.707,149.187
C06821=1182.613,-64.938,-41.862,179.407,5.708,149.188
C06822=1182.618,-65.187,-41.851,179.405,5.707,149.188
C06823=1182.623,-65.437,-41.840,179.402,5.707,149.189
C06824=1182.629,-65.687,-41.828,179.400,5.707,149.190
C06825=1182.634,-65.936,-41.818,179.398,5.706,149.190
C06826=1182.639,-66.186,-41.807,179.396,5.706,149.191
C06827=1182.644,-66.435,-41.796,179.393,5.706,149.191
C06828=1182.650,-66.685,-41.785,179.391,5.706,149.192
C06829=1182.655,-66.935,-41.774,179.389,5.705,149.193
C06830=1182.660,-67.185,-41.763,179.387,5.705,149.193
C06831=1182.665,-67.434,-41.752,179.384,5.705,149.194
C06832=1182.671,-67.684,-41.741,179.382,5.704,149.195
C06833=1182.676,-67.934,-41.730,179.380,5.704,149.195
C06834=1182.681,-68.184,-41.719,179.377,5.704,149.196
C06835=1182.686,-68.433,-41.709,179.375,5.703,149.196
C06836=1182.691,-68.683,-41.698,179.373,5.704,149.197
C06837=1182.697,-68.932,-41.686,179.370,5.703,149.198
C06838=1182.702,-69.183,-41.676,179.368,5.702,149.198
C06839=1182.707,-69.432,-41.665,179.366,5.703,149.199
C06840=1182.712,-69.682,-41.654,179.363,5.702,149.200
C06841=1182.717,-69.931,-41.643,179.361,5.701,149.200
C06842=1182.723,-70.181,-41.633,179.359,5.702,149.201
C06843=1182.728,-70.431,-41.621,179.356,5.701,149.202
C06844=1182.734,-70.680,-41.611,179.354,5.701,149.202
C06845=1182.739,-70.931,-41.600,179.352,5.701,149.203
C06846=1182.744,-71.179,-41.589,179.350,5.700,149.203
C06847=1182.749,-71.430,-41.579,179.347,5.700,149.204
C06848=1182.754,-71.679,-41.567,179.345,5.700,149.205
C06849=1182.759,-71.929,-41.557,179.343,5.699,149.205
C06850=1182.765,-72.179,-41.546,179.340,5.699,149.206
C06851=1182.770,-72.428,-41.535,179.338,5.699,149.207
C06852=1182.775,-72.679,-41.525,179.336,5.699,149.207
C06853=1182.781,-72.928,-41.514,179.333,5.698,149.208
C06854=1182.786,-73.178,-41.503,179.331,5.699,149.209
C06855=1182.791,-73.427,-41.493,179.329,5.698,149.209
C06856=1182.796,-73.677,-41.482,179.327,5.698,149.210
C06857=1182.802,-73.927,-41.471,179.324,5.698,149.210
C06858=1182.807,-74.177,-41.461,179.322,5.697,149.211
C06859=1182.813,-74.426,-41.449,179.320,5.697,149.212
C06860=1182.818,-74.676,-41.439,179.318,5.696,149.212
C06861=1182.823,-74.926,-41.428,179.315,5.696,149.213
C06862=1182.828,-75.175,-41.417,179.313,5.696,149.213
C06863=1182.834,-75.446,-41.407,179.310,5.696,149.214
C06864=1182.839,-75.717,-41.394,179.308,5.695,149.215
C06865=1182.845,-75.989,-41.383,179.305,5.695,149.215
C06866=1182.851,-76.259,-41.372,179.303,5.695,149.216
C06867=1182.856,-76.509,-41.361,179.301,5.695,149.217
C06868=1182.861,-76.758,-41.351,179.298,5.694,149.217
C06869=1182.866,-77.009,-41.340,179.296,5.694,149.218
C06870=1182.872,-77.258,-41.329,179.294,5.694,149.219
C06871=1182.877,-77.508,-41.319,179.291,5.693,149.219
C06872=1182.882,-77.757,-41.308,179.289,5.694,149.220
C06873=1182.887,-78.008,-41.298,179.287,5.693,149.221
C06874=1182.892,-78.256,-41.287,179.285,5.692,149.221
C06875=1182.897,-78.507,-41.276,179.282,5.693,149.222
C06876=1182.903,-78.756,-41.266,179.280,5.692,149.222
C06877=1182.909,-79.006,-41.256,179.278,5.692,149.223
C06878=1182.914,-79.256,-41.245,179.276,5.692,149.224
C06879=1182.919,-79.505,-41.234,179.273,5.691,149.224
C06880=1182.924,-79.755,-41.224,179.271,5.692,149.225
C06881=1182.930,-80.005,-41.214,179.269,5.691,149.226
C06882=1182.935,-80.255,-41.203,179.266,5.690,149.226
C06883=1182.940,-80.505,-41.193,179.264,5.691,149.227
C06884=1182.946,-80.754,-41.183,179.262,5.690,149.227
C06885=1182.950,-81.004,-41.171,179.260,5.690,149.228
C06886=1182.956,-81.253,-41.161,179.257,5.690,149.229
C06887=1182.961,-81.504,-41.151,179.255,5.689,149.229
C06888=1182.967,-81.753,-41.140,179.253,5.690,149.230
C06889=1182.972,-82.003,-41.130,179.250,5.689,149.231
C06890=1182.977,-82.253,-41.120,179.249,5.689,149.231
C06891=1182.983,-82.502,-41.109,179.246,5.689,149.232
C06892=1182.988,-82.753,-41.099,179.244,5.688,149.232
C06893=1182.992,-83.001,-41.088,179.242,5.688,149.233
C06894=1182.997,-83.251,-41.078,179.239,5.688,149.234
C06895=1183.003,-83.501,-41.068,179.237,5.687,149.234
C06896=1183.009,-83.751,-41.058,179.235,5.687,149.235
C06897=1183.014,-84.001,-41.047,179.233,5.687,149.235
C06898=1183.019,-84.250,-41.037,179.231,5.687,149.236
C06899=1183.025,-84.500,-41.027,179.228,5.687,149.237
C06900=1183.030,-84.750,-41.016,179.226,5.686,149.237
C06901=1183.035,-84.999,-41.006,179.224,5.686,149.238
C06902=1183.040,-85.250,-40.996,179.221,5.686,149.239
C06903=1183.045,-85.499,-40.986,179.219,5.686,149.239
C06904=1183.051,-85.749,-40.975,179.217,5.685,149.240
C06905=1183.056,-85.999,-40.965,179.215,5.685,149.240
C06906=1183.061,-86.249,-40.955,179.213,5.685,149.241
C06907=1183.066,-86.498,-40.945,179.210,5.685,149.242
C06908=1183.071,-86.748,-40.934,179.208,5.685,149.242
C06909=1183.077,-86.998,-40.924,179.206,5.684,149.243
C06910=1183.082,-87.247,-40.914,179.203,5.683,149.243
C06911=1183.087,-87.497,-40.903,179.201,5.684,149.244
C06912=1183.092,-87.747,-40.894,179.199,5.683,149.245
C06913=1183.098,-87.996,-40.884,179.197,5.683,149.245
C06914=1183.103,-88.246,-40.873,179.194,5.683,149.246
C06915=1183.109,-88.496,-40.863,179.192,5.682,149.247
C06916=1183.114,-88.745,-40.853,179.190,5.683,149.247
C06917=1183.118,-88.995,-40.843,179.187,5.682,149.248
C06918=1183.124,-89.245,-40.832,179.186,5.682,149.248
C06919=1183.130,-89.494,-40.822,179.183,5.682,149.249
C06920=1183.135,-89.745,-40.812,179.181,5.681,149.250
C06921=1183.140,-89.995,-40.803,179.179,5.681,149.250
C06922=1183.145,-90.244,-40.792,179.177,5.681,149.251
C06923=1183.151,-90.494,-40.782,179.175,5.681,149.252
C06924=1183.156,-90.744,-40.772,179.172,5.681,149.252
C06925=1183.161,-90.993,-40.762,179.170,5.681,149.253
C06926=1183.166,-91.243,-40.752,179.168,5.680,149.253
C06927=1183.171,-91.493,-40.741,179.165,5.679,149.254
C06928=1183.177,-91.742,-40.731,179.163,5.680,149.255
C06929=1183.182,-91.992,-40.722,179.161,5.679,149.255
C06930=1183.188,-92.242,-40.712,179.159,5.679,149.256
C06931=1183.193,-92.492,-40.701,179.156,5.679,149.257
C06932=1183.198,-92.742,-40.691,179.154,5.678,149.257
C06933=1183.203,-92.991,-40.682,179.152,5.679,149.258
C06934=1183.209,-93.240,-40.671,179.150,5.678,149.258
C06935=1183.214,-93.491,-40.662,179.148,5.678,149.259
C06936=1183.219,-93.740,-40.652,179.145,5.678,149.260
C06937=1183.225,-93.990,-40.642,179.144,5.678,149.260
C06938=1183.230,-94.240,-40.631,179.141,5.678,149.261
C06939=1183.235,-94.490,-40.622,179.139,5.677,149.261
C06940=1183.240,-94.740,-40.612,179.137,5.677,149.262
C06941=1183.246,-94.989,-40.602,179.134,5.677,149.263
C06942=1183.251,-95.238,-40.592,179.132,5.677,149.263
C06943=1183.256,-95.489,-40.582,179.130,5.676,149.264
C06944=1183.262,-95.739,-40.572,179.128,5.676,149.264
C06945=1183.267,-95.988,-40.563,179.125,5.676,149.265
C06946=1183.272,-96.238,-40.552,179.123,5.675,149.266
C06947=1183.278,-96.488,-40.543,179.121,5.676,149.266
C06948=1183.282,-96.738,-40.533,179.119,5.675,149.267
C06949=1183.288,-96.987,-40.523,179.117,5.675,149.268
C06950=1183.294,-97.237,-40.512,179.114,5.675,149.268
C06951=1183.299,-97.487,-40.504,179.113,5.675,149.269
C06952=1183.304,-97.736,-40.493,179.110,5.674,149.269
C06953=1183.309,-97.986,-40.483,179.108,5.674,149.270
C06954=1183.314,-98.236,-40.474,179.106,5.674,149.271
C06955=1183.320,-98.486,-40.464,179.103,5.674,149.271
C06956=1183.325,-98.735,-40.454,179.101,5.674,149.272
C06957=1183.331,-98.985,-40.445,179.099,5.673,149.273
C06958=1183.336,-99.234,-40.435,179.097,5.673,149.273
C06959=1183.341,-99.485,-40.424,179.094,5.673,149.274
C06960=1183.347,-99.735,-40.415,179.093,5.673,149.274
C06961=1183.351,-99.984,-40.405,179.090,5.672,149.275
C06962=1183.357,-100.234,-40.395,179.089,5.672,149.275
C06963=1183.362,-100.483,-40.386,179.086,5.672,149.276
C06964=1183.368,-100.733,-40.376,179.083,5.672,149.277
C06965=1183.372,-100.984,-40.367,179.082,5.672,149.277
C06966=1183.378,-101.233,-40.356,179.079,5.671,149.278
C06967=1183.383,-101.505,-40.346,179.077,5.671,149.279
C06968=1183.389,-101.776,-40.336,179.075,5.671,149.279
C06969=1183.395,-102.048,-40.325,179.072,5.671,149.280
C06970=1183.401,-102.320,-40.315,179.070,5.671,149.281
C06971=1183.406,-102.569,-40.305,179.068,5.670,149.281
C06972=1183.412,-102.819,-40.295,179.065,5.670,149.282
C06973=1183.417,-103.068,-40.286,179.063,5.670,149.282
C06974=1183.422,-103.319,-40.276,179.061,5.669,149.283
C06975=1183.427,-103.569,-40.266,179.059,5.669,149.284
C06976=1183.433,-103.819,-40.257,179.057,5.669,149.284
C06977=1183.438,-104.068,-40.247,179.054,5.669,149.285
C06978=1183.443,-104.317,-40.237,179.052,5.669,149.285
C06979=1183.448,-104.567,-40.228,179.050,5.669,149.286
C06980=1183.454,-104.817,-40.218,179.048,5.668,149.287
C06981=1183.459,-105.067,-40.209,179.046,5.669,149.287
C06982=1183.465,-105.316,-40.199,179.044,5.668,149.288
C06983=1183.470,-105.566,-40.190,179.042,5.668,149.289
C06984=1183.476,-105.816,-40.180,179.039,5.667,149.289
C06985=1183.480,-106.066,-40.170,179.037,5.667,149.290
C06986=1183.486,-106.316,-40.161,179.035,5.667,149.290
C06987=1183.491,-106.566,-40.151,179.032,5.667,149.291
C06988=1183.496,-106.815,-40.142,179.031,5.667,149.291
C06989=1183.502,-107.065,-40.132,179.028,5.666,149.292
C06990=1183.507,-107.315,-40.123,179.027,5.666,149.293
C06991=1183.512,-107.564,-40.113,179.024,5.666,149.293
C06992=1183.517,-107.814,-40.104,179.022,5.666,149.294
C06993=1183.523,-108.064,-40.095,179.020,5.666,149.295
C06994=1183.528,-108.314,-40.085,179.018,5.666,149.295
C06995=1183.533,-108.563,-40.076,179.015,5.665,149.296
C06996=1183.539,-108.813,-40.066,179.013,5.666,149.296
C06997=1183.544,-109.063,-40.057,179.011,5.665,149.297
C06998=1183.550,-109.313,-40.048,179.009,5.665,149.298
C06999=1183.555,-109.562,-40.038,179.007,5.664,149.298
C07000=1183.560,-109.812,-40.029,179.005,5.665,149.299
C07001=1183.565,-110.062,-40.019,179.003,5.664,149.299
C07002=1183.570,-110.312,-40.010,179.000,5.665,149.300
C07003=1183.575,-110.562,-40.001,178.998,5.664,149.301
C07004=1183.581,-110.812,-39.991,178.996,5.663,149.301
C07005=1183.586,-111.061,-39.982,178.994,5.663,149.302
C07006=1183.591,-111.311,-39.973,178.991,5.663,149.302
C07007=1183.597,-111.561,-39.963,178.990,5.663,149.303
C07008=1183.602,-111.811,-39.954,178.987,5.663,149.304
C07009=1183.607,-112.061,-39.945,178.985,5.663,149.304
C07010=1183.613,-112.310,-39.935,178.983,5.662,149.305
C07011=1183.618,-112.560,-39.926,178.981,5.662,149.305
C07012=1183.623,-112.810,-39.917,178.978,5.662,149.306
C07013=1183.629,-113.060,-39.907,178.977,5.662,149.307
C07014=1183.634,-113.309,-39.898,178.974,5.661,149.307
C07015=1183.639,-113.559,-39.889,178.973,5.662,149.308
C07016=1183.645,-113.809,-39.879,178.970,5.661,149.308
C07017=1183.650,-114.058,-39.870,178.968,5.661,149.309
C07018=1183.655,-114.308,-39.861,178.966,5.661,149.310
C07019=1183.661,-114.558,-39.851,178.964,5.661,149.310
C07020=1183.666,-114.808,-39.842,178.961,5.660,149.311
C07021=1183.671,-115.058,-39.833,178.960,5.660,149.311
C07022=1183.677,-115.307,-39.824,178.957,5.660,149.312
C07023=1183.683,-115.557,-39.815,178.956,5.660,149.313
C07024=1183.688,-115.807,-39.806,178.953,5.660,149.313
C07025=1183.693,-116.057,-39.797,178.951,5.660,149.314
C07026=1183.699,-116.306,-39.787,178.949,5.659,149.314
C07027=1183.704,-116.556,-39.778,178.947,5.659,149.315
C07028=1183.709,-116.806,-39.769,178.944,5.659,149.316
C07029=1183.714,-117.056,-39.760,178.943,5.659,149.316
C07030=1183.720,-117.306,-39.751,178.940,5.659,149.317
C07031=1183.725,-117.556,-39.742,178.938,5.659,149.317
C07032=1183.730,-117.805,-39.732,178.936,5.658,149.318
C07033=1183.735,-118.055,-39.723,178.934,5.658,149.319
C07034=1183.740,-118.305,-39.714,178.931,5.658,149.319
C07035=1183.746,-118.555,-39.705,178.930,5.658,149.320
C07036=1183.751,-118.805,-39.696,178.927,5.657,149.320
C07037=1183.757,-119.054,-39.687,178.926,5.657,149.321
C07038=1183.762,-119.304,-39.678,178.923,5.657,149.321
C07039=1183.767,-119.553,-39.669,178.921,5.657,149.322
C07040=1183.773,-119.803,-39.659,178.919,5.656,149.323
C07041=1183.778,-120.053,-39.650,178.917,5.657,149.323
C07042=1183.783,-120.303,-39.642,178.915,5.656,149.324
C07043=1183.789,-120.553,-39.633,178.913,5.656,149.325
C07044=1183.794,-120.802,-39.624,178.911,5.656,149.325
C07045=1183.799,-121.052,-39.615,178.908,5.656,149.326
C07046=1183.805,-121.302,-39.605,178.906,5.655,149.326
C07047=1183.810,-121.552,-39.596,178.904,5.656,149.327
C07048=1183.815,-121.802,-39.588,178.902,5.655,149.327
C07049=1183.821,-122.051,-39.579,178.900,5.655,149.328
C07050=1183.826,-122.301,-39.570,178.898,5.655,149.329
C07051=1183.831,-122.550,-39.560,178.896,5.655,149.329
C07052=1183.837,-122.801,-39.551,178.893,5.654,149.330
C07053=1183.842,-123.050,-39.542,178.892,5.654,149.330
C07054=1183.847,-123.300,-39.533,178.889,5.654,149.331
C07055=1183.852,-123.550,-39.524,178.888,5.654,149.332
C07056=1183.858,-123.800,-39.515,178.885,5.653,149.332
C07057=1183.863,-124.049,-39.507,178.883,5.653,149.333
C07058=1183.868,-124.299,-39.498,178.881,5.653,149.333
C07059=1183.874,-124.549,-39.489,178.879,5.653,149.334
C07060=1183.879,-124.799,-39.480,178.877,5.654,149.335
C07061=1183.885,-125.049,-39.471,178.875,5.653,149.335
C07062=1183.890,-125.299,-39.462,178.873,5.653,149.336
C07063=1183.896,-125.548,-39.453,178.870,5.652,149.336
C07064=1183.901,-125.798,-39.444,178.869,5.652,149.337
C07065=1183.906,-126.048,-39.436,178.866,5.652,149.338
C07066=1183.911,-126.298,-39.427,178.865,5.652,149.338
C07067=1183.917,-126.548,-39.418,178.862,5.652,149.339
C07068=1183.922,-126.798,-39.409,178.860,5.652,149.339
C07069=1183.928,-127.047,-39.401,178.858,5.651,149.340
C07070=1183.933,-127.297,-39.392,178.856,5.651,149.340
C07071=1183.512,-127.308,-39.432,178.852,5.655,149.342
C07072=1183.506,-127.058,-39.441,178.854,5.655,149.342
C07073=1183.500,-126.808,-39.449,178.856,5.655,149.341
C07074=1183.495,-126.558,-39.458,178.858,5.655,149.341
C07075=1183.489,-126.309,-39.467,178.861,5.655,149.340
C07076=1183.484,-126.059,-39.476,178.862,5.655,149.339
C07077=1183.479,-125.809,-39.484,178.865,5.656,149.339
C07078=1183.474,-125.559,-39.493,178.867,5.656,149.338
C07079=1183.469,-125.309,-39.502,178.869,5.656,149.338
C07080=1183.464,-125.059,-39.511,178.871,5.656,149.337
C07081=1183.458,-124.810,-39.520,178.873,5.657,149.337
C07082=1183.453,-124.560,-39.529,178.875,5.656,149.336
C07083=1183.448,-124.311,-39.537,178.877,5.657,149.335
C07084=1183.442,-124.061,-39.546,178.879,5.657,149.335
C07085=1183.436,-123.811,-39.556,178.882,5.657,149.334
C07086=1183.431,-123.561,-39.565,178.883,5.657,149.334
C07087=1183.426,-123.311,-39.574,178.886,5.658,149.333
C07088=1183.420,-123.062,-39.582,178.887,5.658,149.332
C07089=1183.415,-122.812,-39.591,178.890,5.658,149.332
C07090=1183.410,-122.562,-39.600,178.892,5.658,149.331
C07091=1183.405,-122.312,-39.609,178.894,5.659,149.331
C07092=1183.400,-122.062,-39.618,178.896,5.659,149.330
C07093=1183.394,-121.812,-39.627,178.898,5.658,149.329
C07094=1183.389,-121.562,-39.636,178.900,5.659,149.329
C07095=1183.383,-121.312,-39.645,178.902,5.658,149.328
C07096=1183.378,-121.063,-39.654,178.905,5.659,149.328
C07097=1183.373,-120.814,-39.663,178.906,5.659,149.327
C07098=1183.368,-120.564,-39.672,178.909,5.660,149.326
C07099=1183.362,-120.314,-39.682,178.910,5.660,149.326
C07100=1183.357,-120.064,-39.690,178.913,5.660,149.325
C07101=1183.351,-119.814,-39.699,178.915,5.660,149.325
C07102=1183.346,-119.564,-39.708,178.917,5.660,149.324
C07103=1183.341,-119.315,-39.717,178.919,5.660,149.324
C07104=1183.336,-119.065,-39.726,178.922,5.661,149.323
C07105=1183.330,-118.815,-39.736,178.923,5.661,149.322
C07106=1183.325,-118.565,-39.744,178.926,5.661,149.322
C07107=1183.319,-118.316,-39.754,178.928,5.661,149.321
C07108=1183.314,-118.066,-39.763,178.930,5.661,149.320
C07109=1183.309,-117.816,-39.772,178.932,5.661,149.320
C07110=1183.303,-117.566,-39.781,178.935,5.662,149.319
C07111=1183.298,-117.316,-39.790,178.936,5.662,149.319
C07112=1183.293,-117.067,-39.799,178.939,5.662,149.318
C07113=1183.288,-116.817,-39.808,178.940,5.662,149.318
C07114=1183.282,-116.567,-39.818,178.943,5.663,149.317
C07115=1183.277,-116.317,-39.827,178.945,5.663,149.316
C07116=1183.272,-116.068,-39.836,178.947,5.663,149.316
C07117=1183.267,-115.818,-39.845,178.949,5.663,149.315
C07118=1183.261,-115.568,-39.855,178.951,5.664,149.315
C07119=1183.256,-115.318,-39.864,178.953,5.663,149.314
C07120=1183.251,-115.068,-39.873,178.955,5.664,149.313
C07121=1183.245,-114.818,-39.882,178.957,5.664,149.313
C07122=1183.240,-114.568,-39.891,178.960,5.664,149.312
C07123=1183.235,-114.319,-39.901,178.962,5.664,149.312
C07124=1183.230,-114.069,-39.909,178.964,5.665,149.311
C07125=1183.224,-113.819,-39.919,178.966,5.664,149.310
C07126=1183.218,-113.569,-39.928,178.968,5.665,149.310
C07127=1183.214,-113.320,-39.938,178.970,5.665,149.309
C07128=1183.208,-113.070,-39.947,178.973,5.665,149.309
C07129=1183.203,-112.820,-39.956,178.975,5.666,149.308
C07130=1183.198,-112.571,-39.966,178.977,5.666,149.307
C07131=1183.192,-112.321,-39.975,178.979,5.666,149.307
C07132=1183.187,-112.071,-39.984,178.981,5.666,149.306
C07133=1183.181,-111.821,-39.993,178.984,5.667,149.306
C07134=1183.176,-111.571,-40.003,178.985,5.667,149.305
C07135=1183.171,-111.322,-40.012,178.988,5.667,149.304
C07136=1183.165,-111.072,-40.021,178.990,5.667,149.304
C07137=1183.160,-110.822,-40.031,178.992,5.667,149.303
C07138=1183.155,-110.572,-40.040,178.994,5.667,149.303
C07139=1183.150,-110.322,-40.049,178.997,5.668,149.302
C07140=1183.144,-110.073,-40.059,178.998,5.668,149.301
C07141=1183.139,-109.823,-40.068,179.001,5.668,149.301
C07142=1183.134,-109.574,-40.078,179.002,5.668,149.300
C07143=1183.128,-109.324,-40.087,179.005,5.668,149.300
C07144=1183.123,-109.074,-40.096,179.007,5.668,149.299
C07145=1183.117,-108.824,-40.106,179.009,5.669,149.298
C07146=1183.112,-108.574,-40.115,179.011,5.668,149.298
C07147=1183.107,-108.325,-40.124,179.014,5.669,149.297
C07148=1183.101,-108.075,-40.134,179.016,5.669,149.296
C07149=1183.096,-107.825,-40.143,179.018,5.670,149.296
C07150=1183.091,-107.576,-40.153,179.020,5.669,149.295
C07151=1183.085,-107.326,-40.162,179.022,5.670,149.295
C07152=1183.081,-107.077,-40.172,179.025,5.670,149.294
C07153=1183.075,-106.826,-40.181,179.026,5.670,149.294
C07154=1183.069,-106.577,-40.190,179.029,5.671,149.293
C07155=1183.064,-106.327,-40.200,179.031,5.671,149.292
C07156=1183.059,-106.076,-40.210,179.033,5.671,149.292
C07157=1183.054,-105.827,-40.220,179.035,5.671,149.291
C07158=1183.049,-105.577,-40.229,179.038,5.671,149.290
C07159=1183.043,-105.328,-40.239,179.039,5.671,149.290
C07160=1183.038,-105.078,-40.248,179.042,5.672,149.289
C07161=1183.033,-104.828,-40.257,179.044,5.672,149.289
C07162=1183.027,-104.578,-40.267,179.046,5.672,149.288
C07163=1183.022,-104.329,-40.277,179.048,5.672,149.288
C07164=1183.016,-104.079,-40.286,179.051,5.673,149.287
C07165=1183.011,-103.830,-40.296,179.053,5.673,149.286
C07166=1183.006,-103.579,-40.306,179.055,5.673,149.286
C07167=1183.001,-103.330,-40.315,179.058,5.673,149.285
C07168=1182.995,-103.079,-40.325,179.059,5.673,149.284
C07169=1182.990,-102.830,-40.334,179.062,5.674,149.284
C07170=1182.985,-102.580,-40.344,179.063,5.674,149.283
C07171=1182.980,-102.331,-40.353,179.066,5.674,149.283
C07172=1182.973,-102.059,-40.364,179.068,5.674,149.282
C07173=1182.968,-101.787,-40.375,179.070,5.675,149.281
C07174=1182.963,-101.515,-40.385,179.073,5.675,149.281
C07175=1182.957,-101.244,-40.395,179.076,5.675,149.280
C07176=1182.951,-100.995,-40.405,179.077,5.675,149.279
C07177=1182.946,-100.744,-40.415,179.080,5.676,149.279
C07178=1182.941,-100.494,-40.425,179.082,5.676,149.278
C07179=1182.935,-100.245,-40.435,179.084,5.676,149.277
C07180=1182.930,-99.995,-40.444,179.086,5.676,149.277
C07181=1182.925,-99.746,-40.454,179.089,5.676,149.276
C07182=1182.920,-99.496,-40.464,179.091,5.676,149.276
C07183=1182.914,-99.245,-40.474,179.093,5.677,149.275
C07184=1182.910,-98.996,-40.483,179.095,5.677,149.274
C07185=1182.904,-98.746,-40.493,179.097,5.677,149.274
C07186=1182.898,-98.496,-40.503,179.100,5.678,149.273
C07187=1182.893,-98.247,-40.513,179.101,5.678,149.273
C07188=1182.887,-97.997,-40.522,179.104,5.678,149.272
C07189=1182.883,-97.747,-40.532,179.106,5.678,149.271
C07190=1182.877,-97.498,-40.542,179.108,5.678,149.271
C07191=1182.871,-97.247,-40.552,179.110,5.678,149.270
C07192=1182.867,-96.998,-40.561,179.113,5.679,149.270
C07193=1182.861,-96.749,-40.572,179.115,5.679,149.269
C07194=1182.856,-96.498,-40.582,179.117,5.679,149.268
C07195=1182.851,-96.249,-40.591,179.119,5.680,149.268
C07196=1182.845,-95.999,-40.601,179.122,5.679,149.267
C07197=1182.840,-95.750,-40.611,179.124,5.680,149.266
C07198=1182.835,-95.500,-40.621,179.126,5.680,149.266
C07199=1182.830,-95.249,-40.631,179.128,5.680,149.265
C07200=1182.825,-95.000,-40.641,179.131,5.681,149.265
C07201=1182.819,-94.751,-40.651,179.132,5.681,149.264
C07202=1182.813,-94.501,-40.661,179.135,5.681,149.263
C07203=1182.809,-94.251,-40.670,179.137,5.681,149.263
C07204=1182.803,-94.001,-40.680,179.139,5.681,149.262
C07205=1182.798,-93.751,-40.691,179.141,5.681,149.261
C07206=1182.793,-93.502,-40.700,179.144,5.682,149.261
C07207=1182.788,-93.251,-40.710,179.146,5.682,149.260
C07208=1182.782,-93.002,-40.720,179.148,5.682,149.260
C07209=1182.776,-92.752,-40.731,179.150,5.683,149.259
C07210=1182.771,-92.503,-40.740,179.153,5.682,149.258
C07211=1182.766,-92.253,-40.751,179.155,5.683,149.258
C07212=1182.761,-92.003,-40.761,179.157,5.683,149.257
C07213=1182.756,-91.753,-40.770,179.159,5.683,149.257
C07214=1182.750,-91.504,-40.780,179.162,5.684,149.256
C07215=1182.745,-91.254,-40.791,179.163,5.684,149.256
C07216=1182.740,-91.004,-40.801,179.166,5.684,149.255
C07217=1182.735,-90.755,-40.810,179.168,5.684,149.254
C07218=1182.730,-90.505,-40.821,179.170,5.685,149.254
C07219=1182.724,-90.255,-40.831,179.173,5.685,149.253
C07220=1182.718,-90.006,-40.841,179.174,5.685,149.252
C07221=1182.713,-89.756,-40.850,179.177,5.685,149.252
C07222=1182.708,-89.505,-40.861,179.179,5.685,149.251
C07223=1182.703,-89.256,-40.871,179.181,5.686,149.251
C07224=1182.697,-89.006,-40.881,179.184,5.686,149.250
C07225=1182.693,-88.756,-40.891,179.186,5.686,149.249
C07226=1182.687,-88.507,-40.902,179.188,5.687,149.249
C07227=1182.682,-88.257,-40.912,179.190,5.686,149.248
C07228=1182.677,-88.007,-40.922,179.193,5.687,149.247
C07229=1182.671,-87.758,-40.933,179.195,5.687,149.247
C07230=1182.666,-87.508,-40.942,179.197,5.687,149.246
C07231=1182.661,-87.258,-40.953,179.200,5.688,149.246
C07232=1182.656,-87.008,-40.963,179.202,5.687,149.245
C07233=1182.650,-86.759,-40.973,179.204,5.688,149.244
C07234=1182.645,-86.509,-40.984,179.206,5.688,149.244
C07235=1182.640,-86.259,-40.993,179.208,5.689,149.243
C07236=1182.635,-86.010,-41.004,179.211,5.689,149.242
C07237=1182.630,-85.760,-41.014,179.213,5.689,149.242
C07238=1182.624,-85.510,-41.024,179.215,5.689,149.241
C07239=1182.618,-85.261,-41.034,179.217,5.689,149.241
C07240=1182.613,-85.010,-41.045,179.219,5.690,149.240
C07241=1182.608,-84.761,-41.055,179.222,5.690,149.239
C07242=1182.603,-84.512,-41.065,179.224,5.690,149.239
C07243=1182.598,-84.261,-41.075,179.226,5.691,149.238
C07244=1182.592,-84.012,-41.086,179.229,5.691,149.237
C07245=1182.587,-83.762,-41.096,179.231,5.691,149.237
C07246=1182.582,-83.512,-41.106,179.233,5.691,149.236
C07247=1182.576,-83.262,-41.117,179.235,5.691,149.236
C07248=1182.571,-83.012,-41.127,179.238,5.692,149.235
C07249=1182.566,-82.763,-41.137,179.240,5.692,149.234
C07250=1182.561,-82.513,-41.147,179.242,5.692,149.234
C07251=1182.556,-82.264,-41.158,179.244,5.693,149.233
C07252=1182.550,-82.014,-41.169,179.247,5.692,149.232
C07253=1182.545,-81.764,-41.179,179.249,5.693,149.232
C07254=1182.540,-81.514,-41.189,179.251,5.693,149.231
C07255=1182.535,-81.264,-41.200,179.253,5.693,149.231
C07256=1182.529,-81.015,-41.210,179.256,5.694,149.230
C07257=1182.524,-80.765,-41.220,179.258,5.694,149.229
C07258=1182.519,-80.515,-41.231,179.260,5.694,149.229
C07259=1182.513,-80.266,-41.242,179.263,5.695,149.228
C07260=1182.508,-80.016,-41.252,179.265,5.694,149.227
C07261=1182.503,-79.766,-41.263,179.267,5.695,149.227
C07262=1182.498,-79.516,-41.273,179.270,5.695,149.226
C07263=1182.492,-79.266,-41.283,179.271,5.695,149.226
C07264=1182.486,-79.017,-41.294,179.274,5.696,149.225
C07265=1182.483,-78.768,-41.304,179.276,5.696,149.224
C07266=1182.477,-78.518,-41.315,179.278,5.696,149.224
C07267=1182.472,-78.268,-41.325,179.281,5.697,149.223
C07268=1182.466,-78.018,-41.335,179.283,5.696,149.222
C07269=1182.462,-77.769,-41.347,179.285,5.697,149.222
C07270=1182.456,-77.519,-41.357,179.288,5.698,149.221
C07271=1182.450,-77.268,-41.368,179.289,5.698,149.221
C07272=1182.445,-77.019,-41.378,179.292,5.698,149.220
C07273=1182.439,-76.770,-41.389,179.295,5.698,149.219
C07274=1182.434,-76.520,-41.400,179.296,5.698,149.219
C07275=1182.429,-76.270,-41.410,179.299,5.699,149.218
C07276=1182.424,-75.999,-41.421,179.302,5.699,149.217
C07277=1182.418,-75.728,-41.433,179.304,5.699,149.217
C07278=1182.411,-75.457,-41.444,179.306,5.699,149.216
C07279=1182.407,-75.186,-41.456,179.309,5.700,149.216
C07280=1182.402,-74.936,-41.466,179.311,5.700,149.215
C07281=1182.396,-74.687,-41.477,179.313,5.700,149.214
C07282=1182.391,-74.437,-41.488,179.315,5.701,149.214
C07283=1182.386,-74.187,-41.498,179.318,5.701,149.213
C07284=1182.380,-73.937,-41.509,179.320,5.701,149.212
C07285=1182.375,-73.688,-41.520,179.322,5.702,149.212
C07286=1182.370,-73.438,-41.531,179.325,5.702,149.211
C07287=1182.364,-73.189,-41.542,179.327,5.702,149.211
C07288=1182.359,-72.939,-41.552,179.329,5.702,149.210
C07289=1182.354,-72.689,-41.563,179.331,5.702,149.209
C07290=1182.349,-72.439,-41.574,179.334,5.703,149.209
C07291=1182.344,-72.190,-41.584,179.336,5.703,149.208
C07292=1182.339,-71.940,-41.595,179.338,5.703,149.207
C07293=1182.333,-71.691,-41.606,179.341,5.704,149.207
C07294=1182.327,-71.440,-41.617,179.343,5.704,149.206
C07295=1182.322,-71.191,-41.628,179.345,5.704,149.205
C07296=1182.317,-70.941,-41.638,179.347,5.705,149.205
C07297=1182.312,-70.691,-41.648,179.350,5.705,149.204
C07298=1182.307,-70.442,-41.660,179.352,5.705,149.204
C07299=1182.301,-70.192,-41.670,179.354,5.705,149.203
C07300=1182.296,-69.942,-41.682,179.357,5.706,149.202
C07301=1182.291,-69.692,-41.692,179.359,5.706,149.202
C07302=1182.286,-69.443,-41.703,179.361,5.706,149.201
C07303=1182.281,-69.193,-41.714,179.364,5.707,149.200
C07304=1182.275,-68.944,-41.725,179.366,5.707,149.200
C07305=1182.270,-68.694,-41.735,179.368,5.707,149.199
C07306=1182.264,-68.444,-41.747,179.371,5.707,149.199
C07307=1182.259,-68.194,-41.757,179.373,5.707,149.198
C07308=1182.255,-67.945,-41.769,179.375,5.708,149.197
C07309=1182.249,-67.695,-41.779,179.378,5.708,149.197
C07310=1182.244,-67.445,-41.790,179.379,5.708,149.196
C07311=1182.238,-67.196,-41.801,179.382,5.709,149.195
C07312=1182.233,-66.946,-41.812,179.385,5.709,149.195
